	        END_IF;
	    END_REGION

	    REGION UNLOADERS & COOLING CONVEYORS
	        IF (#internal.boManSelOnPressL OR #internal.boSetupSelOnPressL OR #internal.boSetupProcActiveL) AND #internal.panel[#PB_Configuration.itLeftSelPbID].boSelect THEN
	            // Enable push-buttons
	            #internal.panel[#PB_Configuration.itUnloaderPbID].boEnable := TRUE;
	            #internal.panel[#PB_Configuration.itUnloaderPCIPbID].boEnable := TRUE;

	            // Modules fault & warning
	            #internal.panel[#PB_Configuration.itUnloaderPbID].boAborted := #EQunloaderL."to".boStatusAbortedEQ OR #EQunloaderL."to".boStatusAbortedSwingInPress OR #EQunloaderL."to".boStatusAbortedUDMove OR #EQunloaderL."to".boStatusAbortedPaddles;
	            #internal.panel[#PB_Configuration.itUnloaderPbID].boHeld := #EQunloaderL."to".boStatusHeldEQ OR #EQunloaderL."to".boStatusHeldSwingInPress OR #EQunloaderL."to".boStatusHeldUDMove OR #EQunloaderL."to".boStatusHeldPaddles;
	            #internal.panel[#PB_Configuration.itUnloaderPCIPbID].boAborted := #EQunloaderL."to".boStatusAbortedEQ OR #EQunloaderL."to".boStatusAbortedSwingInPci OR #EQunloaderL."to".boStatusAbortedExtend;
	            #internal.panel[#PB_Configuration.itUnloaderPCIPbID].boHeld := #EQunloaderL."to".boStatusHeldEQ OR #EQunloaderL."to".boStatusHeldSwingInPci OR #EQunloaderL."to".boStatusHeldExtend;

	            // Unloaders: manual commands
	            IF #internal.panel[#PB_Configuration.itUnloaderPbID].boSelect THEN
	                #internal.panel[#PB_Configuration.itLeftSelPbID].boAborted := #EQunloaderL."to".boStatusAbortedEQ OR #EQunloaderL."to".boStatusAbortedSwingInPress OR #EQunloaderL."to".boStatusAbortedUDMove OR #EQunloaderL."to".boStatusAbortedPaddles;
	                #internal.panel[#PB_Configuration.itLeftSelPbID].boHeld := #EQunloaderL."to".boStatusHeldEQ OR #EQunloaderL."to".boStatusHeldSwingInPress OR #EQunloaderL."to".boStatusHeldUDMove OR #EQunloaderL."to".boStatusHeldPaddles;

	                #internal.panel[#PB_Configuration.itInCmdPbID].boOnPos := #EQunloaderL."to".boPosSwingIn;
	                #internal.panel[#PB_Configuration.itOutCmdPbID].boOnPos := #EQunloaderL."to".boPosSwingOut;
	                #internal.panel[#PB_Configuration.itUpCmdPbID].boOnPos := #EQunloaderL."to".boPosUnloaderUp;
	                #internal.panel[#PB_Configuration.itDownCmdPbID].boOnPos := #EQunloaderL."to".boPosUnloaderDown;
	                #internal.panel[#PB_Configuration.itRetractCmdPbID].boOnPos := #EQunloaderL."to".boPosPaddlesRet;
	                #internal.panel[#PB_Configuration.itExpandCmdPbID].boOnPos := #EQunloaderL."to".boPosPaddlesExp;

	                #internal.panel[#PB_Configuration.itInCmdPbID].boMoving := #EQunloaderL."to".boMoveSwingIn;
	                #internal.panel[#PB_Configuration.itOutCmdPbID].boMoving := #EQunloaderL."to".boMoveSwingOut;
	                #internal.panel[#PB_Configuration.itUpCmdPbID].boMoving := #EQunloaderL."to".boMoveUnloaderUp;
	                #internal.panel[#PB_Configuration.itDownCmdPbID].boMoving := #EQunloaderL."to".boMoveUnloaderDown;
	                #internal.panel[#PB_Configuration.itRetractCmdPbID].boMoving := #EQunloaderL."to".boMovePaddlesRet;
	                #internal.panel[#PB_Configuration.itExpandCmdPbID].boMoving := #EQunloaderL."to".boMovePaddlesExp;

	                #internal.panel[#PB_Configuration.itInCmdPbID].boEnable := #EQunloaderL."to".boEnaSwingIn OR #internal.panel[#PB_Configuration.itInCmdPbID].boOnPos OR #internal.panel[#PB_Configuration.itInCmdPbID].boMoving;
	                #internal.panel[#PB_Configuration.itOutCmdPbID].boEnable := #EQunloaderL."to".boEnaSwingOut OR #internal.panel[#PB_Configuration.itOutCmdPbID].boOnPos OR #internal.panel[#PB_Configuration.itOutCmdPbID].boMoving;
	                #internal.panel[#PB_Configuration.itUpCmdPbID].boEnable := #EQunloaderL."to".boEnaUnloaderUp OR #internal.panel[#PB_Configuration.itUpCmdPbID].boOnPos OR #internal.panel[#PB_Configuration.itUpCmdPbID].boMoving;
	                #internal.panel[#PB_Configuration.itDownCmdPbID].boEnable := #EQunloaderL."to".boEnaUnloaderDown OR #internal.panel[#PB_Configuration.itDownCmdPbID].boOnPos OR #internal.panel[#PB_Configuration.itDownCmdPbID].boMoving;
	                #internal.panel[#PB_Configuration.itRetractCmdPbID].boEnable := #EQunloaderL."to".boEnaPaddlesRet OR #internal.panel[#PB_Configuration.itRetractCmdPbID].boOnPos OR #internal.panel[#PB_Configuration.itRetractCmdPbID].boMoving;
	                #internal.panel[#PB_Configuration.itExpandCmdPbID].boEnable := #EQunloaderL."to".boEnaPaddlesExp OR #internal.panel[#PB_Configuration.itExpandCmdPbID].boOnPos OR #internal.panel[#PB_Configuration.itExpandCmdPbID].boMoving;

	                #EQunloaderL.from.boCmdSwingIn := #internal.panel[#PB_Configuration.itInCmdPbID].boCmdOn;
	                #EQunloaderL.from.boCmdSwingOut := #internal.panel[#PB_Configuration.itOutCmdPbID].boCmdOn;
	                #EQunloaderL.from.boCmdUDMoveDown := #internal.panel[#PB_Configuration.itDownCmdPbID].boCmdOn;
	                #EQunloaderL.from.boCmdUDMoveUp := #internal.panel[#PB_Configuration.itUpCmdPbID].boCmdOn;
	                #EQunloaderL.from.boCmdPaddlesRet := #internal.panel[#PB_Configuration.itRetractCmdPbID].boCmdOn;
	                #EQunloaderL.from.boCmdPaddlesExp := #internal.panel[#PB_Configuration.itExpandCmdPbID].boCmdOn;
	            END_IF;

	            // Unloaders PCI: manual commands
	            IF #internal.panel[#PB_Configuration.itUnloaderPCIPbID].boSelect THEN
	                #internal.panel[#PB_Configuration.itLeftSelPbID].boAborted := #EQunloaderL."to".boStatusAbortedEQ OR #EQunloaderL."to".boStatusAbortedSwingInPress OR #EQunloaderL."to".boStatusAbortedUDMove OR #EQunloaderL."to".boStatusAbortedPaddles;
	                #internal.panel[#PB_Configuration.itLeftSelPbID].boHeld := #EQunloaderL."to".boStatusHeldEQ OR #EQunloaderL."to".boStatusHeldSwingInPress OR #EQunloaderL."to".boStatusHeldUDMove OR #EQunloaderL."to".boStatusHeldPaddles;

	                #internal.panel[#PB_Configuration.itInCmdPbID].boOnPos := #EQunloaderL."to".boPosExtendRet;
	                #internal.panel[#PB_Configuration.itOutCmdPbID].boOnPos := #EQunloaderL."to".boPosExtendExp;
	                #internal.panel[#PB_Configuration.itUpCmdPbID].boOnPos := #EQunloaderL."to".boPosUnloaderUp;
	                #internal.panel[#PB_Configuration.itDownCmdPbID].boOnPos := #EQunloaderL."to".boPosUnloaderDown;
	                #internal.panel[#PB_Configuration.itRetractCmdPbID].boOnPos := #EQunloaderL."to".boPosPaddlesRet;
	                #internal.panel[#PB_Configuration.itExpandCmdPbID].boOnPos := #EQunloaderL."to".boPosPaddlesExp;

	                #internal.panel[#PB_Configuration.itInCmdPbID].boMoving := #EQunloaderL."to".boMoveExtendRet;
	                #internal.panel[#PB_Configuration.itOutCmdPbID].boMoving := #EQunloaderL."to".boMoveExtendExp;
	                #internal.panel[#PB_Configuration.itUpCmdPbID].boMoving := #EQunloaderL."to".boMoveUnloaderUp;
	                #internal.panel[#PB_Configuration.itDownCmdPbID].boMoving := #EQunloaderL."to".boMoveUnloaderDown;
	                #internal.panel[#PB_Configuration.itRetractCmdPbID].boMoving := #EQunloaderL."to".boMovePaddlesRet;
	                #internal.panel[#PB_Configuration.itExpandCmdPbID].boMoving := #EQunloaderL."to".boMovePaddlesExp;

	                #internal.panel[#PB_Configuration.itInCmdPbID].boEnable := #EQunloaderL."to".boEnaExtendRet OR #internal.panel[#PB_Configuration.itInCmdPbID].boOnPos OR #internal.panel[#PB_Configuration.itInCmdPbID].boMoving;
	                #internal.panel[#PB_Configuration.itOutCmdPbID].boEnable := #EQunloaderL."to".boEnaExtendExp OR #internal.panel[#PB_Configuration.itOutCmdPbID].boOnPos OR #internal.panel[#PB_Configuration.itOutCmdPbID].boMoving;
	                #internal.panel[#PB_Configuration.itUpCmdPbID].boEnable := #EQunloaderL."to".boEnaUnloaderUp OR #internal.panel[#PB_Configuration.itUpCmdPbID].boOnPos OR #internal.panel[#PB_Configuration.itUpCmdPbID].boMoving;
	                #internal.panel[#PB_Configuration.itDownCmdPbID].boEnable := #EQunloaderL."to".boEnaUnloaderDown OR #internal.panel[#PB_Configuration.itDownCmdPbID].boOnPos OR #internal.panel[#PB_Configuration.itDownCmdPbID].boMoving;
	                #internal.panel[#PB_Configuration.itRetractCmdPbID].boEnable := #EQunloaderL."to".boEnaPaddlesRet OR #internal.panel[#PB_Configuration.itRetractCmdPbID].boOnPos OR #internal.panel[#PB_Configuration.itRetractCmdPbID].boMoving;
	                #internal.panel[#PB_Configuration.itExpandCmdPbID].boEnable := #EQunloaderL."to".boEnaPaddlesExp OR #internal.panel[#PB_Configuration.itExpandCmdPbID].boOnPos OR #internal.panel[#PB_Configuration.itExpandCmdPbID].boMoving;

	                #EQunloaderL.from.boCmdExtendRet := #internal.panel[#PB_Configuration.itInCmdPbID].boCmdOn;
	                #EQunloaderL.from.boCmdExtendExp := #internal.panel[#PB_Configuration.itOutCmdPbID].boCmdOn;
	                #EQunloaderL.from.boCmdUDMoveDown := #internal.panel[#PB_Configuration.itDownCmdPbID].boCmdOn;
	                #EQunloaderL.from.boCmdUDMoveUp := #internal.panel[#PB_Configuration.itUpCmdPbID].boCmdOn;
	                #EQunloaderL.from.boCmdPaddlesRet := #internal.panel[#PB_Configuration.itRetractCmdPbID].boCmdOn;
	                #EQunloaderL.from.boCmdPaddlesExp := #internal.panel[#PB_Configuration.itExpandCmdPbID].boCmdOn;
	            END_IF;
	        END_IF;
	        IF (#internal.boManSelOnExitConvL OR #internal.boSetupSelOnExitConvL OR #internal.boSetupProcActiveL) AND #internal.panel[#PB_Configuration.itLeftSelPbID].boSelect THEN
	            // Enable push-buttons
	            #internal.panel[#PB_Configuration.itExitConvPbId].boEnable := TRUE;

	            // Modules fault & warning
	            #internal.panel[#PB_Configuration.itExitConvPbId].boAborted := #EQExitConvL."to".boStatusAbortedEQ OR #EQExitConvL."to".boStatusAbortedLwConveyor OR #EQExitConvL."to".boStatusAbortedLwBlocks;
	            #internal.panel[#PB_Configuration.itExitConvPbId].boHeld := #EQExitConvL."to".boStatusHeldEQ OR #EQExitConvL."to".boStatusHeldLwConveyor OR #EQExitConvL."to".boStatusHeldLwBlocks;

	            // Cooling Conveyors : manual commands
	            IF #internal.panel[#PB_Configuration.itExitConvPbId].boSelect THEN
	                #internal.panel[#PB_Configuration.itLeftSelPbID].boAborted := #EQExitConvL."to".boStatusAbortedEQ OR #EQExitConvL."to".boStatusAbortedLwConveyor OR #EQExitConvL."to".boStatusAbortedLwBlocks;
	                #internal.panel[#PB_Configuration.itLeftSelPbID].boHeld := #EQExitConvL."to".boStatusHeldEQ OR #EQExitConvL."to".boStatusHeldLwConveyor OR #EQExitConvL."to".boStatusHeldLwBlocks;

	                #internal.panel[#PB_Configuration.itUpCmdPbID].boOnPos := #EQExitConvL."to".boPosConveyorUp;
	                #internal.panel[#PB_Configuration.itDownCmdPbID].boOnPos := #EQExitConvL."to".boPosConveyorDown;
	                #internal.panel[#PB_Configuration.itOutCmdPbID].boOnPos := FALSE;
	                #internal.panel[#PB_Configuration.itLockCmdPbID].boOnPos := #EQExitConvL."to".boPosBlockIns;
	                #internal.panel[#PB_Configuration.itUnlockCmdPbID].boOnPos := #EQExitConvL."to".boPosBlockRel;

	                #internal.panel[#PB_Configuration.itUpCmdPbID].boMoving := #EQExitConvL."to".boMoveConveyorUp;
	                #internal.panel[#PB_Configuration.itDownCmdPbID].boMoving := #EQExitConvL."to".boMoveConveyorDown;
	                #internal.panel[#PB_Configuration.itOutCmdPbID].boMoving := #EQExitConvL."to".boMoveConveyorFwd;
	                #internal.panel[#PB_Configuration.itLockCmdPbID].boMoving := #EQExitConvL."to".boMoveBlockIns;
	                #internal.panel[#PB_Configuration.itUnlockCmdPbID].boMoving := #EQExitConvL."to".boMoveBlockRel;

	                #internal.panel[#PB_Configuration.itUpCmdPbID].boEnable := #EQExitConvL."to".boEnaConveyorUp OR #internal.panel[#PB_Configuration.itInCmdPbID].boOnPos OR #internal.panel[#PB_Configuration.itInCmdPbID].boMoving;
	                #internal.panel[#PB_Configuration.itDownCmdPbID].boEnable := #EQExitConvL."to".boEnaConveyorDown OR #internal.panel[#PB_Configuration.itInCmdPbID].boOnPos OR #internal.panel[#PB_Configuration.itInCmdPbID].boMoving;
	                #internal.panel[#PB_Configuration.itOutCmdPbID].boEnable := #EQExitConvL."to".boEnaConveyorFwd OR #internal.panel[#PB_Configuration.itInCmdPbID].boOnPos OR #internal.panel[#PB_Configuration.itInCmdPbID].boMoving;
	                #internal.panel[#PB_Configuration.itLockCmdPbID].boEnable := #EQExitConvL."to".boEnaBlockIns OR #internal.panel[#PB_Configuration.itInCmdPbID].boOnPos OR #internal.panel[#PB_Configuration.itInCmdPbID].boMoving;
	                #internal.panel[#PB_Configuration.itUnlockCmdPbID].boEnable := #EQExitConvL."to".boEnaBlockRel OR #internal.panel[#PB_Configuration.itInCmdPbID].boOnPos OR #internal.panel[#PB_Configuration.itInCmdPbID].boMoving;

	                #EQExitConvL.from.boCmdConveyorUp := #internal.panel[#PB_Configuration.itUpCmdPbID].boCmdOn;
	                #EQExitConvL.from.boCmdConveyorDown := #internal.panel[#PB_Configuration.itDownCmdPbID].boCmdOn;
	                #EQExitConvL.from.boCmdConveyorFwd := #internal.panel[#PB_Configuration.itOutCmdPbID].boCmdOn;
	                #EQExitConvL.from.boCmdBlockIns := #internal.panel[#PB_Configuration.itLockCmdPbID].boCmdOn;
	                #EQExitConvL.from.boCmdBlockRel := #internal.panel[#PB_Configuration.itUnlockCmdPbID].boCmdOn;
	            END_IF;
	        END_IF;

	        IF (#internal.boManSelOnPressR OR #internal.boSetupSelOnPressR OR #internal.boSetupProcActiveR) AND #internal.panel[#PB_Configuration.itRightSelPbID].boSelect THEN
	            // Enable push-buttons
	            #internal.panel[#PB_Configuration.itUnloaderPbID].boEnable := TRUE;
	            #internal.panel[#PB_Configuration.itUnloaderPCIPbID].boEnable := TRUE;

	            // Modules fault & warning
	            #internal.panel[#PB_Configuration.itUnloaderPbID].boAborted := #EQunloaderR."to".boStatusAbortedEQ OR #EQunloaderR."to".boStatusAbortedSwingInPress OR #EQunloaderR."to".boStatusAbortedUDMove OR #EQunloaderR."to".boStatusAbortedPaddles;
	            #internal.panel[#PB_Configuration.itUnloaderPbID].boHeld := #EQunloaderR."to".boStatusHeldEQ OR #EQunloaderR."to".boStatusHeldSwingInPress OR #EQunloaderR."to".boStatusHeldUDMove OR #EQunloaderR."to".boStatusHeldPaddles;
	            #internal.panel[#PB_Configuration.itUnloaderPCIPbID].boAborted := #EQunloaderR."to".boStatusAbortedEQ OR #EQunloaderR."to".boStatusAbortedSwingInPci OR #EQunloaderR."to".boStatusAbortedExtend;
	            #internal.panel[#PB_Configuration.itUnloaderPCIPbID].boHeld := #EQunloaderR."to".boStatusHeldEQ OR #EQunloaderR."to".boStatusHeldSwingInPci OR #EQunloaderR."to".boStatusHeldExtend;

	            // Unloaders: manual commands
	            IF #internal.panel[#PB_Configuration.itUnloaderPbID].boSelect THEN
	                #internal.panel[#PB_Configuration.itRightSelPbID].boAborted := #EQunloaderR."to".boStatusAbortedEQ OR #EQunloaderR."to".boStatusAbortedSwingInPress OR #EQunloaderR."to".boStatusAbortedUDMove OR #EQunloaderR."to".boStatusAbortedPaddles;
	                #internal.panel[#PB_Configuration.itRightSelPbID].boHeld := #EQunloaderR."to".boStatusHeldEQ OR #EQunloaderR."to".boStatusHeldSwingInPress OR #EQunloaderR."to".boStatusHeldUDMove OR #EQunloaderR."to".boStatusHeldPaddles;

	                #internal.panel[#PB_Configuration.itInCmdPbID].boOnPos := #EQunloaderR."to".boPosSwingIn;
	                #internal.panel[#PB_Configuration.itOutCmdPbID].boOnPos := #EQunloaderR."to".boPosSwingOut;
	                #internal.panel[#PB_Configuration.itUpCmdPbID].boOnPos := #EQunloaderR."to".boPosUnloaderUp;
	                #internal.panel[#PB_Configuration.itDownCmdPbID].boOnPos := #EQunloaderR."to".boPosUnloaderDown;
	                #internal.panel[#PB_Configuration.itRetractCmdPbID].boOnPos := #EQunloaderR."to".boPosPaddlesRet;
	                #internal.panel[#PB_Configuration.itExpandCmdPbID].boOnPos := #EQunloaderR."to".boPosPaddlesExp;

	                #internal.panel[#PB_Configuration.itInCmdPbID].boMoving := #EQunloaderR."to".boMoveSwingIn;
	                #internal.panel[#PB_Configuration.itOutCmdPbID].boMoving := #EQunloaderR."to".boMoveSwingOut;
	                #internal.panel[#PB_Configuration.itUpCmdPbID].boMoving := #EQunloaderR."to".boMoveUnloaderUp;
	                #internal.panel[#PB_Configuration.itDownCmdPbID].boMoving := #EQunloaderR."to".boMoveUnloaderDown;
	                #internal.panel[#PB_Configuration.itRetractCmdPbID].boMoving := #EQunloaderR."to".boMovePaddlesRet;
	                #internal.panel[#PB_Configuration.itExpandCmdPbID].boMoving := #EQunloaderR."to".boMovePaddlesExp;

	                #internal.panel[#PB_Configuration.itInCmdPbID].boEnable := #EQunloaderR."to".boEnaSwingIn OR #internal.panel[#PB_Configuration.itInCmdPbID].boOnPos OR #internal.panel[#PB_Configuration.itInCmdPbID].boMoving;
	                #internal.panel[#PB_Configuration.itOutCmdPbID].boEnable := #EQunloaderR."to".boEnaSwingOut OR #internal.panel[#PB_Configuration.itOutCmdPbID].boOnPos OR #internal.panel[#PB_Configuration.itOutCmdPbID].boMoving;
	                #internal.panel[#PB_Configuration.itUpCmdPbID].boEnable := #EQunloaderR."to".boEnaUnloaderUp OR #internal.panel[#PB_Configuration.itUpCmdPbID].boOnPos OR #internal.panel[#PB_Configuration.itUpCmdPbID].boMoving;
	                #internal.panel[#PB_Configuration.itDownCmdPbID].boEnable := #EQunloaderR."to".boEnaUnloaderDown OR #internal.panel[#PB_Configuration.itDownCmdPbID].boOnPos OR #internal.panel[#PB_Configuration.itDownCmdPbID].boMoving;
	                #internal.panel[#PB_Configuration.itRetractCmdPbID].boEnable := #EQunloaderR."to".boEnaPaddlesRet OR #internal.panel[#PB_Configuration.itRetractCmdPbID].boOnPos OR #internal.panel[#PB_Configuration.itRetractCmdPbID].boMoving;
	                #internal.panel[#PB_Configuration.itExpandCmdPbID].boEnable := #EQunloaderR."to".boEnaPaddlesExp OR #internal.panel[#PB_Configuration.itExpandCmdPbID].boOnPos OR #internal.panel[#PB_Configuration.itExpandCmdPbID].boMoving;

	                #EQunloaderR.from.boCmdSwingIn := #internal.panel[#PB_Configuration.itInCmdPbID].boCmdOn;
	                #EQunloaderR.from.boCmdSwingOut := #internal.panel[#PB_Configuration.itOutCmdPbID].boCmdOn;
	                #EQunloaderR.from.boCmdUDMoveDown := #internal.panel[#PB_Configuration.itDownCmdPbID].boCmdOn;
	                #EQunloaderR.from.boCmdUDMoveUp := #internal.panel[#PB_Configuration.itUpCmdPbID].boCmdOn;
	                #EQunloaderR.from.boCmdPaddlesRet := #internal.panel[#PB_Configuration.itRetractCmdPbID].boCmdOn;
	                #EQunloaderR.from.boCmdPaddlesExp := #internal.panel[#PB_Configuration.itExpandCmdPbID].boCmdOn;
	            END_IF;

	            // Unloaders PCI: manual commands
	            IF #internal.panel[#PB_Configuration.itUnloaderPCIPbID].boSelect THEN
	                #internal.panel[#PB_Configuration.itRightSelPbID].boAborted := #EQunloaderR."to".boStatusAbortedEQ OR #EQunloaderR."to".boStatusAbortedSwingInPci OR #EQunloaderR."to".boStatusAbortedExtend;
	                #internal.panel[#PB_Configuration.itRightSelPbID].boHeld := #EQunloaderR."to".boStatusHeldEQ OR #EQunloaderR."to".boStatusHeldSwingInPci OR #EQunloaderR."to".boStatusHeldExtend;

	                #internal.panel[#PB_Configuration.itInCmdPbID].boOnPos := #EQunloaderR."to".boPosExtendRet;
	                #internal.panel[#PB_Configuration.itOutCmdPbID].boOnPos := #EQunloaderR."to".boPosExtendExp;
	                #internal.panel[#PB_Configuration.itUpCmdPbID].boOnPos := #EQunloaderR."to".boPosUnloaderUp;
	                #internal.panel[#PB_Configuration.itDownCmdPbID].boOnPos := #EQunloaderR."to".boPosUnloaderDown;
	                #internal.panel[#PB_Configuration.itRetractCmdPbID].boOnPos := #EQunloaderR."to".boPosPaddlesRet;
	                #internal.panel[#PB_Configuration.itExpandCmdPbID].boOnPos := #EQunloaderR."to".boPosPaddlesExp;

	                #internal.panel[#PB_Configuration.itInCmdPbID].boMoving := #EQunloaderR."to".boMoveExtendRet;
	                #internal.panel[#PB_Configuration.itOutCmdPbID].boMoving := #EQunloaderR."to".boMoveExtendExp;
	                #internal.panel[#PB_Configuration.itUpCmdPbID].boMoving := #EQunloaderR."to".boMoveUnloaderUp;
	                #internal.panel[#PB_Configuration.itDownCmdPbID].boMoving := #EQunloaderR."to".boMoveUnloaderDown;
	                #internal.panel[#PB_Configuration.itRetractCmdPbID].boMoving := #EQunloaderR."to".boMovePaddlesRet;
	                #internal.panel[#PB_Configuration.itExpandCmdPbID].boMoving := #EQunloaderR."to".boMovePaddlesExp;

	                #internal.panel[#PB_Configuration.itInCmdPbID].boEnable := #EQunloaderR."to".boEnaExtendRet OR #internal.panel[#PB_Configuration.itInCmdPbID].boOnPos OR #internal.panel[#PB_Configuration.itInCmdPbID].boMoving;
	                #internal.panel[#PB_Configuration.itOutCmdPbID].boEnable := #EQunloaderR."to".boEnaExtendExp OR #internal.panel[#PB_Configuration.itOutCmdPbID].boOnPos OR #internal.panel[#PB_Configuration.itOutCmdPbID].boMoving;
	                #internal.panel[#PB_Configuration.itUpCmdPbID].boEnable := #EQunloaderR."to".boEnaUnloaderUp OR #internal.panel[#PB_Configuration.itUpCmdPbID].boOnPos OR #internal.panel[#PB_Configuration.itUpCmdPbID].boMoving;
	                #internal.panel[#PB_Configuration.itDownCmdPbID].boEnable := #EQunloaderR."to".boEnaUnloaderDown OR #internal.panel[#PB_Configuration.itDownCmdPbID].boOnPos OR #internal.panel[#PB_Configuration.itDownCmdPbID].boMoving;
	                #internal.panel[#PB_Configuration.itRetractCmdPbID].boEnable := #EQunloaderR."to".boEnaPaddlesRet OR #internal.panel[#PB_Configuration.itRetractCmdPbID].boOnPos OR #internal.panel[#PB_Configuration.itRetractCmdPbID].boMoving;
	                #internal.panel[#PB_Configuration.itExpandCmdPbID].boEnable := #EQunloaderR."to".boEnaPaddlesExp OR #internal.panel[#PB_Configuration.itExpandCmdPbID].boOnPos OR #internal.panel[#PB_Configuration.itExpandCmdPbID].boMoving;

	                #EQunloaderR.from.boCmdExtendRet := #internal.panel[#PB_Configuration.itInCmdPbID].boCmdOn;
	                #EQunloaderR.from.boCmdExtendExp := #internal.panel[#PB_Configuration.itOutCmdPbID].boCmdOn;
	                #EQunloaderR.from.boCmdUDMoveDown := #internal.panel[#PB_Configuration.itDownCmdPbID].boCmdOn;
	                #EQunloaderR.from.boCmdUDMoveUp := #internal.panel[#PB_Configuration.itUpCmdPbID].boCmdOn;
	                #EQunloaderR.from.boCmdPaddlesRet := #internal.panel[#PB_Configuration.itRetractCmdPbID].boCmdOn;
	                #EQunloaderR.from.boCmdPaddlesExp := #internal.panel[#PB_Configuration.itExpandCmdPbID].boCmdOn;
	            END_IF;
	        END_IF;
	        IF (#internal.boManSelOnExitConvR OR #internal.boSetupSelOnExitConvR OR #internal.boSetupProcActiveR) AND #internal.panel[#PB_Configuration.itRightSelPbID].boSelect THEN

	            // Enable push-buttons
	            #internal.panel[#PB_Configuration.itExitConvPbId].boEnable := TRUE;

	            // Modules fault & warning
	            #internal.panel[#PB_Configuration.itExitConvPbId].boAborted := #EQExitConvR."to".boStatusAbortedEQ OR #EQExitConvR."to".boStatusAbortedLwConveyor OR #EQExitConvR."to".boStatusAbortedLwBlocks;
	            #internal.panel[#PB_Configuration.itExitConvPbId].boHeld := #EQExitConvR."to".boStatusHeldEQ OR #EQExitConvR."to".boStatusHeldLwConveyor OR #EQExitConvR."to".boStatusHeldLwBlocks;

	            // Cooling Conveyors : manual commands
	            IF #internal.panel[#PB_Configuration.itExitConvPbId].boSelect THEN
	                #internal.panel[#PB_Configuration.itRightSelPbID].boAborted := #EQExitConvR."to".boStatusAbortedEQ OR #EQExitConvR."to".boStatusAbortedLwConveyor OR #EQExitConvR."to".boStatusAbortedLwBlocks;
	                #internal.panel[#PB_Configuration.itRightSelPbID].boHeld := #EQExitConvR."to".boStatusHeldEQ OR #EQExitConvR."to".boStatusHeldLwConveyor OR #EQExitConvR."to".boStatusHeldLwBlocks;

	                #internal.panel[#PB_Configuration.itUpCmdPbID].boOnPos := #EQExitConvR."to".boPosConveyorUp;
	                #internal.panel[#PB_Configuration.itDownCmdPbID].boOnPos := #EQExitConvR."to".boPosConveyorDown;
	                #internal.panel[#PB_Configuration.itOutCmdPbID].boOnPos := FALSE;
	                #internal.panel[#PB_Configuration.itLockCmdPbID].boOnPos := #EQExitConvR."to".boPosBlockIns;
	                #internal.panel[#PB_Configuration.itUnlockCmdPbID].boOnPos := #EQExitConvR."to".boPosBlockRel;

	                #internal.panel[#PB_Configuration.itUpCmdPbID].boMoving := #EQExitConvR."to".boMoveConveyorUp;
	                #internal.panel[#PB_Configuration.itDownCmdPbID].boMoving := #EQExitConvR."to".boMoveConveyorDown;
	                #internal.panel[#PB_Configuration.itOutCmdPbID].boMoving := #EQExitConvR."to".boMoveConveyorFwd;
	                #internal.panel[#PB_Configuration.itLockCmdPbID].boMoving := #EQExitConvR."to".boMoveBlockIns;
	                #internal.panel[#PB_Configuration.itUnlockCmdPbID].boMoving := #EQExitConvR."to".boMoveBlockRel;

	                #internal.panel[#PB_Configuration.itUpCmdPbID].boEnable := #EQExitConvR."to".boEnaConveyorUp OR #internal.panel[#PB_Configuration.itInCmdPbID].boOnPos OR #internal.panel[#PB_Configuration.itInCmdPbID].boMoving;
	                #internal.panel[#PB_Configuration.itDownCmdPbID].boEnable := #EQExitConvR."to".boEnaConveyorDown OR #internal.panel[#PB_Configuration.itInCmdPbID].boOnPos OR #internal.panel[#PB_Configuration.itInCmdPbID].boMoving;
	                #internal.panel[#PB_Configuration.itOutCmdPbID].boEnable := #EQExitConvR."to".boEnaConveyorFwd OR #internal.panel[#PB_Configuration.itInCmdPbID].boOnPos OR #internal.panel[#PB_Configuration.itInCmdPbID].boMoving;
	                #internal.panel[#PB_Configuration.itLockCmdPbID].boEnable := #EQExitConvR."to".boEnaBlockIns OR #internal.panel[#PB_Configuration.itInCmdPbID].boOnPos OR #internal.panel[#PB_Configuration.itInCmdPbID].boMoving;
	                #internal.panel[#PB_Configuration.itUnlockCmdPbID].boEnable := #EQExitConvR."to".boEnaBlockRel OR #internal.panel[#PB_Configuration.itInCmdPbID].boOnPos OR #internal.panel[#PB_Configuration.itInCmdPbID].boMoving;

	                #EQExitConvR.from.boCmdConveyorUp := #internal.panel[#PB_Configuration.itUpCmdPbID].boCmdOn;
	                #EQExitConvR.from.boCmdConveyorDown := #internal.panel[#PB_Configuration.itDownCmdPbID].boCmdOn;
	                #EQExitConvR.from.boCmdConveyorFwd := #internal.panel[#PB_Configuration.itOutCmdPbID].boCmdOn;
	                #EQExitConvR.from.boCmdBlockIns := #internal.panel[#PB_Configuration.itLockCmdPbID].boCmdOn;
	                #EQExitConvR.from.boCmdBlockRel := #internal.panel[#PB_Configuration.itUnlockCmdPbID].boCmdOn;
	            END_IF;

	        END_IF;

	        IF ((#internal.boManSelOnPressL OR #internal.boSetupSelOnPressL OR #internal.boSetupProcActiveL) AND #internal.panel[#PB_Configuration.itLeftSelPbID].boSelect) AND
	            ((#internal.boManSelOnPressR OR #internal.boSetupSelOnPressR OR #internal.boSetupProcActiveR) AND #internal.panel[#PB_Configuration.itRightSelPbID].boSelect) THEN
	            // Enable push-buttons
	            #internal.panel[#PB_Configuration.itUnloaderPbID].boEnable := TRUE;
	            #internal.panel[#PB_Configuration.itUnloaderPCIPbID].boEnable := TRUE;

	            // Modules fault & warning
	            #internal.panel[#PB_Configuration.itUnloaderPbID].boAborted := #EQunloaderL."to".boStatusAbortedEQ OR #EQunloaderL."to".boStatusAbortedSwingInPress OR #EQunloaderL."to".boStatusAbortedUDMove OR #EQunloaderL."to".boStatusAbortedPaddles OR
	            #EQunloaderR."to".boStatusAbortedEQ OR #EQunloaderR."to".boStatusAbortedSwingInPress OR #EQunloaderR."to".boStatusAbortedUDMove OR #EQunloaderR."to".boStatusAbortedPaddles;
	            #internal.panel[#PB_Configuration.itUnloaderPbID].boHeld := #EQunloaderL."to".boStatusHeldEQ OR #EQunloaderL."to".boStatusHeldSwingInPress OR #EQunloaderL."to".boStatusHeldUDMove OR #EQunloaderL."to".boStatusHeldPaddles OR
	            #EQunloaderR."to".boStatusHeldEQ OR #EQunloaderR."to".boStatusHeldSwingInPress OR #EQunloaderR."to".boStatusHeldUDMove OR #EQunloaderR."to".boStatusHeldPaddles;

	            #internal.panel[#PB_Configuration.itUnloaderPCIPbID].boAborted := #EQunloaderL."to".boStatusAbortedEQ OR #EQunloaderL."to".boStatusAbortedSwingInPci OR #EQunloaderL."to".boStatusAbortedExtend OR
	            #EQunloaderR."to".boStatusAbortedEQ OR #EQunloaderR."to".boStatusAbortedSwingInPci OR #EQunloaderR."to".boStatusAbortedExtend;
	            #internal.panel[#PB_Configuration.itUnloaderPCIPbID].boHeld := #EQunloaderL."to".boStatusHeldEQ OR #EQunloaderL."to".boStatusHeldSwingInPci OR #EQunloaderL."to".boStatusHeldExtend OR
	            #EQunloaderR."to".boStatusHeldEQ OR #EQunloaderR."to".boStatusHeldSwingInPci OR #EQunloaderR."to".boStatusHeldExtend;

	            // Unloaders: manual commands
	            IF #internal.panel[#PB_Configuration.itUnloaderPbID].boSelect THEN
	                #internal.panel[#PB_Configuration.itInCmdPbID].boOnPos := #EQunloaderL."to".boPosSwingIn AND #EQunloaderR."to".boPosSwingIn;
	                #internal.panel[#PB_Configuration.itOutCmdPbID].boOnPos := #EQunloaderL."to".boPosSwingOut AND #EQunloaderR."to".boPosSwingOut;
	                #internal.panel[#PB_Configuration.itUpCmdPbID].boOnPos := #EQunloaderL."to".boPosUnloaderUp AND #EQunloaderR."to".boPosUnloaderUp;
	                #internal.panel[#PB_Configuration.itDownCmdPbID].boOnPos := #EQunloaderL."to".boPosUnloaderDown AND #EQunloaderR."to".boPosUnloaderDown;
	                #internal.panel[#PB_Configuration.itRetractCmdPbID].boOnPos := #EQunloaderL."to".boPosPaddlesRet AND #EQunloaderR."to".boPosPaddlesRet;
	                #internal.panel[#PB_Configuration.itExpandCmdPbID].boOnPos := #EQunloaderL."to".boPosPaddlesExp AND #EQunloaderR."to".boPosPaddlesExp;

	                #internal.panel[#PB_Configuration.itInCmdPbID].boMoving := #EQunloaderL."to".boMoveSwingIn AND #EQunloaderR."to".boMoveSwingIn;
	                #internal.panel[#PB_Configuration.itOutCmdPbID].boMoving := #EQunloaderL."to".boMoveSwingOut AND #EQunloaderR."to".boMoveSwingOut;
	                #internal.panel[#PB_Configuration.itUpCmdPbID].boMoving := #EQunloaderL."to".boMoveUnloaderUp AND #EQunloaderR."to".boMoveUnloaderUp;
	                #internal.panel[#PB_Configuration.itDownCmdPbID].boMoving := #EQunloaderL."to".boMoveUnloaderDown AND #EQunloaderR."to".boMoveUnloaderDown;
	                #internal.panel[#PB_Configuration.itRetractCmdPbID].boMoving := #EQunloaderL."to".boMovePaddlesRet AND #EQunloaderR."to".boMovePaddlesRet;
	                #internal.panel[#PB_Configuration.itExpandCmdPbID].boMoving := #EQunloaderL."to".boMovePaddlesExp AND #EQunloaderR."to".boMovePaddlesExp;

	                #internal.panel[#PB_Configuration.itInCmdPbID].boEnable := #EQunloaderL."to".boEnaSwingIn OR #EQunloaderR."to".boEnaSwingIn OR #internal.panel[#PB_Configuration.itInCmdPbID].boOnPos OR #internal.panel[#PB_Configuration.itInCmdPbID].boMoving;
	                #internal.panel[#PB_Configuration.itOutCmdPbID].boEnable := #EQunloaderL."to".boEnaSwingOut OR #EQunloaderR."to".boEnaSwingOut OR #internal.panel[#PB_Configuration.itOutCmdPbID].boOnPos OR #internal.panel[#PB_Configuration.itOutCmdPbID].boMoving;
	                #internal.panel[#PB_Configuration.itUpCmdPbID].boEnable := #EQunloaderL."to".boEnaUnloaderUp OR #EQunloaderR."to".boEnaUnloaderUp OR #internal.panel[#PB_Configuration.itUpCmdPbID].boOnPos OR #internal.panel[#PB_Configuration.itUpCmdPbID].boMoving;
	                #internal.panel[#PB_Configuration.itDownCmdPbID].boEnable := #EQunloaderL."to".boEnaUnloaderDown OR #EQunloaderR."to".boEnaUnloaderDown OR #internal.panel[#PB_Configuration.itDownCmdPbID].boOnPos OR #internal.panel[#PB_Configuration.itDownCmdPbID].boMoving;
	                #internal.panel[#PB_Configuration.itRetractCmdPbID].boEnable := #EQunloaderL."to".boEnaPaddlesRet OR #EQunloaderR."to".boEnaPaddlesRet OR #internal.panel[#PB_Configuration.itRetractCmdPbID].boOnPos OR #internal.panel[#PB_Configuration.itRetractCmdPbID].boMoving;
	                #internal.panel[#PB_Configuration.itExpandCmdPbID].boEnable := #EQunloaderL."to".boEnaPaddlesExp OR #EQunloaderR."to".boEnaPaddlesExp OR #internal.panel[#PB_Configuration.itExpandCmdPbID].boOnPos OR #internal.panel[#PB_Configuration.itExpandCmdPbID].boMoving;
	            END_IF;

	            // Unloaders PCI: manual commands
	            IF #internal.panel[#PB_Configuration.itUnloaderPCIPbID].boSelect THEN
	                #internal.panel[#PB_Configuration.itInCmdPbID].boOnPos := #EQunloaderL."to".boPosExtendRet AND #EQunloaderR."to".boPosExtendRet;
	                #internal.panel[#PB_Configuration.itOutCmdPbID].boOnPos := #EQunloaderL."to".boPosExtendExp AND #EQunloaderR."to".boPosExtendExp;
	                #internal.panel[#PB_Configuration.itUpCmdPbID].boOnPos := #EQunloaderL."to".boPosUnloaderUp AND #EQunloaderR."to".boPosUnloaderUp;
	                #internal.panel[#PB_Configuration.itDownCmdPbID].boOnPos := #EQunloaderL."to".boPosUnloaderDown AND #EQunloaderR."to".boPosUnloaderDown;
	                #internal.panel[#PB_Configuration.itRetractCmdPbID].boOnPos := #EQunloaderL."to".boPosPaddlesRet AND #EQunloaderR."to".boPosPaddlesRet;
	                #internal.panel[#PB_Configuration.itExpandCmdPbID].boOnPos := #EQunloaderL."to".boPosPaddlesExp AND #EQunloaderR."to".boPosPaddlesExp;

	                #internal.panel[#PB_Configuration.itInCmdPbID].boMoving := #EQunloaderL."to".boMoveExtendRet OR #EQunloaderR."to".boMoveExtendRet;
	                #internal.panel[#PB_Configuration.itOutCmdPbID].boMoving := #EQunloaderL."to".boMoveExtendExp OR #EQunloaderR."to".boMoveExtendExp;
	                #internal.panel[#PB_Configuration.itUpCmdPbID].boMoving := #EQunloaderL."to".boMoveUnloaderUp AND #EQunloaderR."to".boMoveUnloaderUp;
	                #internal.panel[#PB_Configuration.itDownCmdPbID].boMoving := #EQunloaderL."to".boMoveUnloaderDown AND #EQunloaderR."to".boMoveUnloaderDown;
	                #internal.panel[#PB_Configuration.itRetractCmdPbID].boMoving := #EQunloaderL."to".boMovePaddlesRet OR #EQunloaderR."to".boMovePaddlesRet;
	                #internal.panel[#PB_Configuration.itExpandCmdPbID].boMoving := #EQunloaderL."to".boMovePaddlesExp OR #EQunloaderR."to".boMovePaddlesExp;

	                #internal.panel[#PB_Configuration.itInCmdPbID].boEnable := #EQunloaderL."to".boEnaExtendRet OR #EQunloaderR."to".boEnaExtendRet OR #internal.panel[#PB_Configuration.itInCmdPbID].boOnPos OR #internal.panel[#PB_Configuration.itInCmdPbID].boMoving;
	                #internal.panel[#PB_Configuration.itOutCmdPbID].boEnable := #EQunloaderL."to".boEnaExtendExp OR #EQunloaderR."to".boEnaExtendExp OR #internal.panel[#PB_Configuration.itOutCmdPbID].boOnPos OR #internal.panel[#PB_Configuration.itOutCmdPbID].boMoving;
	                #internal.panel[#PB_Configuration.itUpCmdPbID].boEnable := #EQunloaderL."to".boEnaUnloaderUp OR #EQunloaderR."to".boEnaUnloaderUp OR #internal.panel[#PB_Configuration.itUpCmdPbID].boOnPos OR #internal.panel[#PB_Configuration.itUpCmdPbID].boMoving;
	                #internal.panel[#PB_Configuration.itDownCmdPbID].boEnable := #EQunloaderL."to".boEnaUnloaderDown OR #EQunloaderR."to".boEnaUnloaderDown OR #internal.panel[#PB_Configuration.itDownCmdPbID].boOnPos OR #internal.panel[#PB_Configuration.itDownCmdPbID].boMoving;
	                #internal.panel[#PB_Configuration.itRetractCmdPbID].boEnable := #EQunloaderL."to".boEnaPaddlesRet OR #EQunloaderR."to".boEnaPaddlesRet OR #internal.panel[#PB_Configuration.itRetractCmdPbID].boOnPos OR #internal.panel[#PB_Configuration.itRetractCmdPbID].boMoving;
	                #internal.panel[#PB_Configuration.itExpandCmdPbID].boEnable := #EQunloaderL."to".boEnaPaddlesExp OR #EQunloaderR."to".boEnaPaddlesExp OR #internal.panel[#PB_Configuration.itExpandCmdPbID].boOnPos OR #internal.panel[#PB_Configuration.itExpandCmdPbID].boMoving;
	            END_IF;


	            // Enable push-buttons
	            #internal.panel[#PB_Configuration.itExitConvPbId].boEnable := TRUE;

	            // Modules fault & warning
	            #internal.panel[#PB_Configuration.itExitConvPbId].boAborted := #EQExitConvL."to".boStatusAbortedEQ OR #EQExitConvL."to".boStatusAbortedLwConveyor OR #EQExitConvL."to".boStatusAbortedLwBlocks OR
	            #EQExitConvR."to".boStatusAbortedEQ OR #EQExitConvR."to".boStatusAbortedLwConveyor OR #EQExitConvR."to".boStatusAbortedLwBlocks;
	            #internal.panel[#PB_Configuration.itExitConvPbId].boHeld := #EQExitConvL."to".boStatusHeldEQ OR #EQExitConvL."to".boStatusHeldLwConveyor OR #EQExitConvL."to".boStatusHeldLwBlocks OR
	            #EQExitConvR."to".boStatusHeldEQ OR #EQExitConvR."to".boStatusHeldLwConveyor OR #EQExitConvR."to".boStatusHeldLwBlocks;

	            // Cooling Conveyors : manual commands
	            IF #internal.panel[#PB_Configuration.itExitConvPbId].boSelect THEN
	                #internal.panel[#PB_Configuration.itRightSelPbID].boAborted := #EQExitConvL."to".boStatusAbortedEQ OR #EQExitConvL."to".boStatusAbortedLwConveyor OR #EQExitConvL."to".boStatusAbortedLwBlocks OR
	                #EQExitConvR."to".boStatusAbortedEQ OR #EQExitConvR."to".boStatusAbortedLwConveyor OR #EQExitConvR."to".boStatusAbortedLwBlocks;
	                #internal.panel[#PB_Configuration.itRightSelPbID].boHeld := #EQExitConvL."to".boStatusHeldEQ OR #EQExitConvL."to".boStatusHeldLwConveyor OR #EQExitConvL."to".boStatusHeldLwBlocks OR
	                #EQExitConvR."to".boStatusHeldEQ OR #EQExitConvR."to".boStatusHeldLwConveyor OR #EQExitConvR."to".boStatusHeldLwBlocks;

	                #internal.panel[#PB_Configuration.itUpCmdPbID].boOnPos := #EQExitConvL."to".boPosConveyorUp AND #EQExitConvR."to".boPosLwConveyorUp;
	                #internal.panel[#PB_Configuration.itDownCmdPbID].boOnPos := #EQExitConvL."to".boPosConveyorDown AND #EQExitConvR."to".boPosLwConveyorDown;
	                #internal.panel[#PB_Configuration.itOutCmdPbID].boOnPos := FALSE;
	                #internal.panel[#PB_Configuration.itLockCmdPbID].boOnPos := #EQExitConvL."to".boPosBlockIns AND #EQExitConvR."to".boPosLwBlockIns;
	                #internal.panel[#PB_Configuration.itUnlockCmdPbID].boOnPos := #EQExitConvL."to".boPosBlockRel AND #EQExitConvR."to".boPosLwBlockRel;

	                #internal.panel[#PB_Configuration.itUpCmdPbID].boMoving := #EQExitConvR."to".boMoveConveyorUp OR #EQExitConvR."to".boMoveLwConveyorUp;
	                #internal.panel[#PB_Configuration.itDownCmdPbID].boMoving := #EQExitConvR."to".boMoveConveyorDown OR #EQExitConvR."to".boMoveLwConveyorDown;
	                #internal.panel[#PB_Configuration.itOutCmdPbID].boMoving := #EQExitConvR."to".boMoveConveyorFwd OR #EQExitConvR."to".boMoveLwConveyorFwd;
	                #internal.panel[#PB_Configuration.itLockCmdPbID].boMoving := #EQExitConvR."to".boMoveBlockIns OR #EQExitConvR."to".boMoveLwBlockIns;
	                #internal.panel[#PB_Configuration.itUnlockCmdPbID].boMoving := #EQExitConvR."to".boMoveBlockRel OR #EQExitConvR."to".boMoveLwBlockRel;

	                #internal.panel[#PB_Configuration.itUpCmdPbID].boEnable := #EQExitConvL."to".boEnaConveyorUp OR #EQExitConvR."to".boEnaLwConveyorUp OR #internal.panel[#PB_Configuration.itInCmdPbID].boOnPos OR #internal.panel[#PB_Configuration.itInCmdPbID].boMoving;
	                #internal.panel[#PB_Configuration.itDownCmdPbID].boEnable := #EQExitConvL."to".boEnaConveyorDown OR #EQExitConvR."to".boEnaLwConveyorDown OR #internal.panel[#PB_Configuration.itInCmdPbID].boOnPos OR #internal.panel[#PB_Configuration.itInCmdPbID].boMoving;
	                #internal.panel[#PB_Configuration.itOutCmdPbID].boEnable := #EQExitConvL."to".boEnaConveyorFwd OR #EQExitConvR."to".boEnaLwConveyorFwd OR #internal.panel[#PB_Configuration.itInCmdPbID].boOnPos OR #internal.panel[#PB_Configuration.itInCmdPbID].boMoving;
	                #internal.panel[#PB_Configuration.itLockCmdPbID].boEnable := #EQExitConvL."to".boEnaBlockIns OR #EQExitConvR."to".boEnaLwBlockIns OR #internal.panel[#PB_Configuration.itInCmdPbID].boOnPos OR #internal.panel[#PB_Configuration.itInCmdPbID].boMoving;
	                #internal.panel[#PB_Configuration.itUnlockCmdPbID].boEnable := #EQExitConvL."to".boEnaBlockRel OR #EQExitConvR."to".boEnaLwBlockRel OR #internal.panel[#PB_Configuration.itInCmdPbID].boOnPos OR #internal.panel[#PB_Configuration.itInCmdPbID].boMoving;
	            END_IF;

	        END_IF;
	    END_REGION

	END_REGION

	//=======================================================================================================================================
	//            PRODUCTION PROGRAM AUTO
	//=======================================================================================================================================
	REGION PRODUCTION PROGRAM AUTO
	   REGION LEFT
	        IF #internal.boAutoSelOnPressL THEN
	            #internal.panel[#PB_Configuration.itLeftSelPbID].boAborted := #EQgtsL."to".boStatusAbortedEQ OR #EQloaderL."to".boStatusAbortedEQ OR #EQcenterMechL."to".boStatusAbortedEQ OR #EQintHeatL."to".boStatusAbortedEQ OR
	            #EQpressL."to".boStatusAbortedEQ OR #EQextHeatL."to".boStatusAbortedEQ OR #EQunloaderL."to".boStatusAbortedEQ OR #EQExitConvL."to".boStatusAbortedEQ;
	            #internal.panel[#PB_Configuration.itLeftSelPbID].boHeld := #EQgtsL."to".boStatusHeldEQ OR #EQloaderL."to".boStatusHeldEQ OR #EQcenterMechL."to".boStatusHeldEQ OR #EQintHeatL."to".boStatusHeldEQ OR #EQpressL."to".boStatusHeldEQ OR
	            #EQextHeatL."to".boStatusHeldEQ OR #EQunloaderL."to".boStatusHeldEQ OR #EQExitConvL."to".boStatusHeldEQ OR #unitL."to".boMoldDisabled OR #unitL."to".boLoadDisabled;
	            IF #internal.panel[#PB_Configuration.itLeftSelPbID].boSelect THEN
	                REGION LOADER & MGTS & UNIT
	                    #internal.panel[#PB_Configuration.itLoaderPbID].boEnable := TRUE;
	                    #internal.panel[#PB_Configuration.itGTSPbID].boEnable := TRUE;

	                    IF NOT #internal.panel[#PB_Configuration.itRightSelPbID].boSelect THEN
	                        // Modules fault & warning
	                        #internal.panel[#PB_Configuration.itGTSPbID].boAborted := #EQgtsL."to".boStatusAbortedEQ;
	                        #internal.panel[#PB_Configuration.itGTSPbID].boHeld := #EQgtsL."to".boStatusHeldEQ;
	                        #internal.panel[#PB_Configuration.itLoaderPbID].boAborted := #EQloaderL."to".boStatusAbortedEQ;
	                        #internal.panel[#PB_Configuration.itLoaderPbID].boHeld := #EQloaderL."to".boStatusHeldEQ OR #unitL."to".boLoadDisabled;
	                    END_IF;

	                    // MGTS: automatic command
	                    IF #internal.panel[#PB_Configuration.itGTSPbID].boSelect THEN
	                        #internal.panel[#PB_Configuration.itOnOffSelPbID].boEnable := TRUE;
	                    END_IF;

	                    // Loaders: automatic command
	                    IF #internal.panel[#PB_Configuration.itLoaderPbID].boSelect THEN
	                        #internal.panel[#PB_Configuration.itOnOffSelPbID].boEnable := TRUE;
	                        // Protection for wrong disable timer
	                        #internal.disableFilterLeft(IN := #internal.panel[#PB_Configuration.itOnOffSelPbID].boCmdOn AND NOT #internal.boDisableEQLmem,
	                                                   PT := T#2s,
	                                                   Q => #internal.boDisableEQLmem);

	                        IF #internal.boDisableEQLmem AND #internal.panel[#PB_Configuration.itLeftSelPbID].boSelect THEN
	                            #unitL.from.boLoadDisableReq := TRUE;
	                        END_IF;
	                    END_IF;

	                    // Unit procedure commands: pick-up
	                    #internal.panel[#PB_Configuration.itUnitPbID].boEnable := #internal.panel[#PB_Configuration.itUnitPbID].boAborted OR #internal.panel[#PB_Configuration.itUnitPbID].boHeld;
	                    #internal.panel[#PB_Configuration.itPickupPbID].boEnable := #unitL."to".boEnaPickUp OR #internal.panel[#PB_Configuration.itPickupPbID].boAborted; //AND internal.panel[itLeftSelPbID].boSelect;

	                    // Modules fault & warning
	                    #internal.panel[#PB_Configuration.itUnitPbID].boAborted := #unitL."to".boStatusAbortedEQ;
	                    #internal.panel[#PB_Configuration.itPickupPbID].boAborted := #unitL."to".boRescueTireOccured;
	                    #internal.panel[#PB_Configuration.itUnitPbID].boHeld := #unitL."to".boStatusHeldEQ;

	                    // Pick-up command
	                    IF #internal.panel[#PB_Configuration.itPickupPbID].boSelect THEN
	                        #internal.panel[#PB_Configuration.itOnOffSelPbID].boEnable := TRUE;
	                        #internal.panel[#PB_Configuration.itLeftSelPbID].boSelect := #unitL."to".boEnaPickUp AND NOT #unitL."to".boLoadDisabled;
	                        #unitL.from.boPickUpCmd := #internal.panel[#PB_Configuration.itOnOffSelPbID].boCmdRE AND #internal.panel[#PB_Configuration.itLeftSelPbID].boSelect AND #unitL."to".boEnaPickUp AND NOT #unitL."to".boLoadDisabled;
	                    END_IF;

	                END_REGION

	                REGION PRESSES
	                    #internal.panel[#PB_Configuration.itPressPbID].boEnable := TRUE;

	                    IF NOT #internal.panel[#PB_Configuration.itRightSelPbID].boSelect THEN
	                        // Modules fault & warning
	                        #internal.panel[#PB_Configuration.itPressPbID].boAborted := #EQpressL."to".boStatusAbortedEQ;
	                        #internal.panel[#PB_Configuration.itPressPbID].boHeld := #EQpressL."to".boStatusHeldEQ OR #unitL."to".boMoldDisabled;
	                    END_IF;

	                    // Press: automatic commands
	                    IF #internal.panel[#PB_Configuration.itPressPbID].boSelect THEN
	                        #internal.panel[#PB_Configuration.itOnOffSelPbID].boEnable := TRUE;
	                        IF #internal.panel[#PB_Configuration.itOnOffSelPbID].boCmdRE AND FALSE THEN
	                            #unitL.from.boMoldDisableReq := TRUE;
	                        END_IF;
	                    END_IF;
	                END_REGION

	                REGION CENTER-MECH
	                    #internal.panel[#PB_Configuration.itTopRingPbID].boEnable := TRUE;// internal.panel[itTopRingPbID].boAborted OR internal.panel[itTopRingPbID].boHeld;
	                    #internal.panel[#PB_Configuration.itBotRingPbID].boEnable := TRUE;// internal.panel[itBotRingPbID].boAborted OR internal.panel[itBotRingPbID].boHeld;
	                    #internal.panel[#PB_Configuration.itBeadRingPbID].boEnable := TRUE;// internal.panel[itBeadRingPbID].boAborted OR internal.panel[itBeadRingPbID].boHeld;

	                    IF NOT #internal.panel[#PB_Configuration.itRightSelPbID].boSelect THEN
	                        // Modules fault & warning
	                        #internal.panel[#PB_Configuration.itTopRingPbID].boAborted := #EQcenterMechL."to".boStatusAbortedEQ OR #EQcenterMechL."to".boStatusAbortedTCRing;
	                        #internal.panel[#PB_Configuration.itTopRingPbID].boHeld := #EQcenterMechL."to".boStatusHeldEQ OR #EQcenterMechL."to".boStatusHeldTCRing;
	                        #internal.panel[#PB_Configuration.itBotRingPbID].boAborted := #EQcenterMechL."to".boStatusAbortedEQ OR #EQcenterMechL."to".boStatusAbortedBCRing;
	                        #internal.panel[#PB_Configuration.itBotRingPbID].boHeld := #EQcenterMechL."to".boStatusHeldEQ OR #EQcenterMechL."to".boStatusHeldBCRing;
	                        #internal.panel[#PB_Configuration.itBeadRingPbID].boAborted := #EQcenterMechL."to".boStatusAbortedEQ OR #EQcenterMechL."to".boStatusAbortedBeadRing;
	                        #internal.panel[#PB_Configuration.itBeadRingPbID].boHeld := #EQcenterMechL."to".boStatusHeldEQ OR #EQcenterMechL."to".boStatusHeldBeadRing;
	                    END_IF;
	                    // Top Ring: automatic commands
	                    IF #internal.panel[#PB_Configuration.itTopRingPbID].boSelect THEN
	                        #internal.panel[#PB_Configuration.itOnOffSelPbID].boEnable := TRUE;
	                    END_IF;
	                    // Bottom Ring: automatic commands
	                    IF #internal.panel[#PB_Configuration.itBotRingPbID].boSelect THEN
	                        #internal.panel[#PB_Configuration.itOnOffSelPbID].boEnable := TRUE;
	                    END_IF;
	                    // Bead Ring: automatic commands
	                    IF #internal.panel[#PB_Configuration.itBeadRingPbID].boSelect THEN
	                        #internal.panel[#PB_Configuration.itOnOffSelPbID].boEnable := TRUE;
	                    END_IF;
	                END_REGION

	                REGION UNLOADER & COOLING CONVEYORS
	                #internal.panel[#PB_Configuration.itUnloaderPbID].boEnable := TRUE;
	                #internal.panel[#PB_Configuration.itUnloaderPCIPbID].boEnable := TRUE;
	                #internal.panel[#PB_Configuration.itExitConvPbId].boEnable := TRUE;

	                IF NOT #internal.panel[#PB_Configuration.itRightSelPbID].boSelect THEN
	                    // Modules fault & warning
	                    #internal.panel[#PB_Configuration.itUnloaderPbID].boAborted := #EQunloaderL."to".boStatusAbortedEQ;
	                    #internal.panel[#PB_Configuration.itUnloaderPbID].boHeld := #EQunloaderL."to".boStatusHeldEQ;
	                    #internal.panel[#PB_Configuration.itUnloaderPCIPbID].boAborted := #EQunloaderL."to".boStatusAbortedEQ;
	                    #internal.panel[#PB_Configuration.itUnloaderPCIPbID].boHeld := #EQunloaderL."to".boStatusHeldEQ;
	                    #internal.panel[#PB_Configuration.itExitConvPbId].boAborted := #EQExitConvL."to".boStatusAbortedEQ;
	                    #internal.panel[#PB_Configuration.itExitConvPbId].boHeld := #EQExitConvL."to".boStatusHeldEQ;
	                END_IF;
	                // Unloader: automatic commands
	                IF #internal.panel[#PB_Configuration.itUnloaderPbID].boSelect OR #internal.panel[#PB_Configuration.itUnloaderPCIPbID].boSelect THEN
	                    #internal.panel[#PB_Configuration.itOnOffSelPbID].boEnable := TRUE;
	                    IF #internal.panel[#PB_Configuration.itOnOffSelPbID].boCmdRE THEN
	                        #unitL.from.boUnloadDisableReq := TRUE;
	                    END_IF;
	                END_IF;

	                // Cooling conveyors: automatic commands
	                IF #internal.panel[#PB_Configuration.itExitConvPbId].boSelect THEN
	                    #internal.panel[#PB_Configuration.itOnOffSelPbID].boEnable := TRUE;
	                END_IF;
	            END_REGION
	        END_IF;
	        END_IF;
	    END_REGION

	    REGION RIGHT
	    IF #internal.boAutoSelOnPressR THEN
	        #internal.panel[#PB_Configuration.itRightSelPbID].boAborted := #EQgtsR."to".boStatusAbortedEQ OR #EQloaderR."to".boStatusAbortedEQ OR #EQcenterMechR."to".boStatusAbortedEQ OR #EQintHeatR."to".boStatusAbortedEQ OR
	        #EQpressR."to".boStatusAbortedEQ OR #EQextHeatR."to".boStatusAbortedEQ OR #EQunloaderR."to".boStatusAbortedEQ OR #EQExitConvR."to".boStatusAbortedEQ;
	        #internal.panel[#PB_Configuration.itRightSelPbID].boHeld := #EQgtsR."to".boStatusHeldEQ OR #EQloaderR."to".boStatusHeldEQ OR #EQcenterMechR."to".boStatusHeldEQ OR #EQintHeatR."to".boStatusHeldEQ OR #EQpressR."to".boStatusHeldEQ OR
	        #EQextHeatR."to".boStatusHeldEQ OR #EQunloaderR."to".boStatusHeldEQ OR #EQExitConvR."to".boStatusHeldEQ OR #unitR."to".boMoldDisabled OR #unitR."to".boLoadDisabled;


	        IF #internal.panel[#PB_Configuration.itRightSelPbID].boSelect THEN
	            REGION LOADER & MGTS & UNIT
	                #internal.panel[#PB_Configuration.itLoaderPbID].boEnable := TRUE;
	                #internal.panel[#PB_Configuration.itGTSPbID].boEnable := TRUE;

	                IF NOT #internal.panel[#PB_Configuration.itLeftSelPbID].boSelect THEN
	                    // Modules fault & warning
	                    #internal.panel[#PB_Configuration.itGTSPbID].boAborted := #EQgtsR."to".boStatusAbortedEQ;
	                    #internal.panel[#PB_Configuration.itGTSPbID].boHeld := #EQgtsR."to".boStatusHeldEQ;
	                    #internal.panel[#PB_Configuration.itLoaderPbID].boAborted := #EQloaderR."to".boStatusAbortedEQ;
	                    #internal.panel[#PB_Configuration.itLoaderPbID].boHeld := #EQloaderR."to".boStatusHeldEQ OR #unitR."to".boLoadDisabled;
	                END_IF;

	                // MGTS: automatic command
	                IF #internal.panel[#PB_Configuration.itGTSPbID].boSelect THEN
	                    #internal.panel[#PB_Configuration.itOnOffSelPbID].boEnable := TRUE;
	                END_IF;

	                // Loaders: automatic command
	                IF #internal.panel[#PB_Configuration.itLoaderPbID].boSelect THEN
	                    #internal.panel[#PB_Configuration.itOnOffSelPbID].boEnable := TRUE;

	                    // Protection for wrong disable timer
	                    #internal.disableFilterRight(IN := #internal.panel[#PB_Configuration.itOnOffSelPbID].boCmdOn AND NOT #internal.boDisableEQRmem,
	                                                 PT := T#2s,
	                                                 Q => #internal.boDisableEQRmem);

	                    IF #internal.boDisableEQRmem AND #internal.panel[#PB_Configuration.itRightSelPbID].boSelect THEN
	                        #unitR.from.boLoadDisableReq := TRUE;
	                    END_IF;
	                END_IF;

	                // Unit procedure commands: pick-up
	                #internal.panel[#PB_Configuration.itUnitPbID].boEnable := #internal.panel[#PB_Configuration.itUnitPbID].boAborted OR #internal.panel[#PB_Configuration.itUnitPbID].boHeld;
	                #internal.panel[#PB_Configuration.itPickupPbID].boEnable := #unitR."to".boEnaPickUp OR #internal.panel[#PB_Configuration.itPickupPbID].boAborted; //AND internal.panel[itRightSelPbID].boSelect;

	                // Modules fault & warning
	                #internal.panel[#PB_Configuration.itUnitPbID].boAborted := #unitR."to".boStatusAbortedEQ;
	                #internal.panel[#PB_Configuration.itPickupPbID].boAborted := #unitR."to".boRescueTireOccured;
	                #internal.panel[#PB_Configuration.itUnitPbID].boHeld := #unitR."to".boStatusHeldEQ;

	                // Pick-up command
	                IF #internal.panel[#PB_Configuration.itPickupPbID].boSelect THEN
	                    #internal.panel[#PB_Configuration.itOnOffSelPbID].boEnable := TRUE;
	                    #internal.panel[#PB_Configuration.itRightSelPbID].boSelect := #unitR."to".boEnaPickUp AND NOT #unitR."to".boLoadDisabled;
	                    #unitR.from.boPickUpCmd := #internal.panel[#PB_Configuration.itOnOffSelPbID].boCmdRE AND #internal.panel[#PB_Configuration.itRightSelPbID].boSelect AND #unitR."to".boEnaPickUp AND NOT #unitR."to".boLoadDisabled;
	                END_IF;
	            END_REGION
	            REGION PRESSES
	                #internal.panel[#PB_Configuration.itPressPbID].boEnable := TRUE;

	                IF NOT #internal.panel[#PB_Configuration.itLeftSelPbID].boSelect THEN
	                    // Modules fault & warning
	                    #internal.panel[#PB_Configuration.itPressPbID].boAborted := #EQpressR."to".boStatusAbortedEQ;
	                    #internal.panel[#PB_Configuration.itPressPbID].boHeld := #EQpressR."to".boStatusHeldEQ OR #unitR."to".boMoldDisabled;
	                END_IF;

	                // Press: automatic commands
	                IF #internal.panel[#PB_Configuration.itPressPbID].boSelect THEN
	                    #internal.panel[#PB_Configuration.itOnOffSelPbID].boEnable := TRUE;
	                    IF #internal.panel[#PB_Configuration.itOnOffSelPbID].boCmdRE AND FALSE THEN
	                        #unitR.from.boMoldDisableReq := TRUE;
	                    END_IF;
	                END_IF;
	            END_REGION
	            REGION CENTER-MECH
	                #internal.panel[#PB_Configuration.itTopRingPbID].boEnable := TRUE;// internal.panel[itTopRingPbID].boAborted OR internal.panel[itTopRingPbID].boHeld;
	                #internal.panel[#PB_Configuration.itBotRingPbID].boEnable := TRUE;// internal.panel[itBotRingPbID].boAborted OR internal.panel[itBotRingPbID].boHeld;
	                #internal.panel[#PB_Configuration.itBeadRingPbID].boEnable := TRUE;// internal.panel[itBeadRingPbID].boAborted OR internal.panel[itBeadRingPbID].boHeld;

	                IF NOT #internal.panel[#PB_Configuration.itLeftSelPbID].boSelect THEN
	                    // Modules fault & warning
	                    #internal.panel[#PB_Configuration.itTopRingPbID].boAborted := #EQcenterMechR."to".boStatusAbortedEQ OR #EQcenterMechR."to".boStatusAbortedTCRing;
	                    #internal.panel[#PB_Configuration.itTopRingPbID].boHeld := #EQcenterMechR."to".boStatusHeldEQ OR #EQcenterMechR."to".boStatusHeldTCRing;
	                    #internal.panel[#PB_Configuration.itBotRingPbID].boAborted := #EQcenterMechR."to".boStatusAbortedEQ OR #EQcenterMechR."to".boStatusAbortedBCRing;
	                    #internal.panel[#PB_Configuration.itBotRingPbID].boHeld := #EQcenterMechR."to".boStatusHeldEQ OR #EQcenterMechR."to".boStatusHeldBCRing;
	                    #internal.panel[#PB_Configuration.itBeadRingPbID].boAborted := #EQcenterMechR."to".boStatusAbortedEQ OR #EQcenterMechR."to".boStatusAbortedBeadRing;
	                    #internal.panel[#PB_Configuration.itBeadRingPbID].boHeld := #EQcenterMechR."to".boStatusHeldEQ OR #EQcenterMechR."to".boStatusHeldBeadRing;
	                END_IF;

	                // Top Ring: automatic commands
	                IF #internal.panel[#PB_Configuration.itTopRingPbID].boSelect THEN
	                    #internal.panel[#PB_Configuration.itOnOffSelPbID].boEnable := TRUE;
	                END_IF;
	                // Bottom Ring: automatic commands
	                IF #internal.panel[#PB_Configuration.itBotRingPbID].boSelect THEN
	                    #internal.panel[#PB_Configuration.itOnOffSelPbID].boEnable := TRUE;
	                END_IF;
	                // Bead Ring: automatic commands
	                IF #internal.panel[#PB_Configuration.itBeadRingPbID].boSelect THEN
	                    #internal.panel[#PB_Configuration.itOnOffSelPbID].boEnable := TRUE;
	                END_IF;
	            END_REGION
	            REGION UNLOADER & COOLING CONVEYORS
	                #internal.panel[#PB_Configuration.itUnloaderPbID].boEnable := TRUE;
	                #internal.panel[#PB_Configuration.itUnloaderPCIPbID].boEnable := TRUE;
	                #internal.panel[#PB_Configuration.itExitConvPbId].boEnable := TRUE;

	                IF NOT #internal.panel[#PB_Configuration.itLeftSelPbID].boSelect THEN
	                    // Modules fault & warning
	                    #internal.panel[#PB_Configuration.itUnloaderPbID].boAborted := #EQunloaderR."to".boStatusAbortedEQ;
	                    #internal.panel[#PB_Configuration.itUnloaderPbID].boHeld := #EQunloaderR."to".boStatusHeldEQ;
	                    #internal.panel[#PB_Configuration.itUnloaderPCIPbID].boAborted := #EQunloaderR."to".boStatusAbortedEQ;
	                    #internal.panel[#PB_Configuration.itUnloaderPCIPbID].boHeld := #EQunloaderR."to".boStatusHeldEQ;
	                    #internal.panel[#PB_Configuration.itExitConvPbId].boAborted := #EQExitConvR."to".boStatusAbortedEQ;
	                    #internal.panel[#PB_Configuration.itExitConvPbId].boHeld := #EQExitConvR."to".boStatusHeldEQ;
	                END_IF;

	                // Unloader: automatic commands
	                IF #internal.panel[#PB_Configuration.itUnloaderPbID].boSelect OR #internal.panel[#PB_Configuration.itUnloaderPCIPbID].boSelect THEN
	                    #internal.panel[#PB_Configuration.itOnOffSelPbID].boEnable := TRUE;
	                    IF #internal.panel[#PB_Configuration.itOnOffSelPbID].boCmdRE THEN
	                        #unitR.from.boUnloadDisableReq := TRUE;
	                    END_IF;
	                END_IF;

	                IF #internal.panel[#PB_Configuration.itExitConvPbId].boSelect THEN
	                    #internal.panel[#PB_Configuration.itOnOffSelPbID].boEnable := TRUE;
	                END_IF;
	            END_REGION
	        END_IF;
	    END_IF;
	END_REGION

	    REGION HEATING (INTERNAL & EXTERNAL)
	    IF #internal.boAutoSelOnHeatingL THEN
	        #internal.panel[#PB_Configuration.itShapingPbID].boEnable := TRUE;
	        #internal.panel[#PB_Configuration.itExtHeatingPbID].boEnable := TRUE;

	        IF NOT #internal.panel[#PB_Configuration.itRightSelPbID].boSelect THEN
	            // Unit curing active
	            #internal.panel[#PB_Configuration.itShapingPbID].boMoving := #EQintHeatL."to".boCuringActive;

	            // Unit procedure commands: gym
	            #internal.panel[#PB_Configuration.itGymPbID].boEnable := #unitL."to".boEnaGym OR #unitL."to".boGymActivated;
	            #internal.panel[#PB_Configuration.itGymPbID].boHeld := #unitL."to".boGymActivated AND NOT #internal.panel[#PB_Configuration.itGymPbID].boSelect;
	            #internal.panel[#PB_Configuration.itExtHeatingPbID].boHeld := NOT #unitL."to".boMoldPrewarmDone AND NOT #unitL."to".boMoldDisabled;

	            // External heating pre-warm done
	            #internal.panel[#PB_Configuration.itLeftSelPbID].boHeld := NOT #unitL."to".boMoldPrewarmDone AND NOT #unitL."to".boMoldDisabled;
	        END_IF;

	        IF #internal.panel[#PB_Configuration.itGymPbID].boSelect THEN
	            #internal.panel[#PB_Configuration.itOnOffSelPbID].boEnable := TRUE;
	            #unitL.from.boGymCmd := #internal.panel[#PB_Configuration.itLeftSelPbID].boSelect AND #internal.panel[#PB_Configuration.itOnOffSelPbID].boCmdRE;
	        END_IF;

	    END_IF;

	    IF #internal.boAutoSelOnHeatingR THEN
	        #internal.panel[#PB_Configuration.itShapingPbID].boEnable := TRUE;
	        #internal.panel[#PB_Configuration.itExtHeatingPbID].boEnable := TRUE;

	        IF NOT #internal.panel[#PB_Configuration.itLeftSelPbID].boSelect THEN
	            // Unit curing active
	            #internal.panel[#PB_Configuration.itShapingPbID].boMoving := #EQintHeatR."to".boCuringActive;

	            // Unit procedure commands: gym
	            #internal.panel[#PB_Configuration.itGymPbID].boEnable := #unitR."to".boEnaGym OR #unitR."to".boGymActivated;
	            #internal.panel[#PB_Configuration.itGymPbID].boHeld := #unitR."to".boGymActivated AND NOT #internal.panel[#PB_Configuration.itGymPbID].boSelect;
	            #internal.panel[#PB_Configuration.itExtHeatingPbID].boHeld := NOT #unitR."to".boMoldPrewarmDone AND NOT #unitR."to".boMoldDisabled;

	            // External heating pre-warm done
	            #internal.panel[#PB_Configuration.itRightSelPbID].boHeld := NOT #unitR."to".boMoldPrewarmDone AND NOT #unitR."to".boMoldDisabled;
	        END_IF;

	        IF #internal.panel[#PB_Configuration.itGymPbID].boSelect THEN
	            #internal.panel[#PB_Configuration.itOnOffSelPbID].boEnable := TRUE;
	            #unitR.from.boGymCmd := #internal.panel[#PB_Configuration.itRightSelPbID].boSelect AND #internal.panel[#PB_Configuration.itOnOffSelPbID].boCmdRE;
	        END_IF;
	    END_IF;

	    IF #internal.boAutoSelOnHeatingL AND #internal.panel[#PB_Configuration.itLeftSelPbID].boSelect AND
	        #internal.boAutoSelOnHeatingR AND #internal.panel[#PB_Configuration.itRightSelPbID].boSelect THEN
	        // Unit curing active
	        #internal.panel[#PB_Configuration.itShapingPbID].boMoving := #EQintHeatL."to".boCuringActive OR #EQintHeatR."to".boCuringActive;
	        // Unit procedure commands: gym
	        #internal.panel[#PB_Configuration.itGymPbID].boEnable := #unitL."to".boEnaGym OR #unitL."to".boGymActivated OR #unitR."to".boEnaGym OR #unitR."to".boGymActivated;
	        #internal.panel[#PB_Configuration.itGymPbID].boHeld := (#unitL."to".boGymActivated OR #unitR."to".boGymActivated) AND NOT #internal.panel[#PB_Configuration.itGymPbID].boSelect;
	        #internal.panel[#PB_Configuration.itExtHeatingPbID].boHeld := (NOT #unitL."to".boMoldPrewarmDone AND NOT #unitL."to".boMoldDisabled) OR (NOT #unitR."to".boMoldPrewarmDone AND NOT #unitR."to".boMoldDisabled);

	        // External heating pre-warm done
	        #internal.panel[#PB_Configuration.itLeftSelPbID].boHeld := NOT #unitL."to".boMoldPrewarmDone AND NOT #unitL."to".boMoldDisabled;
	        #internal.panel[#PB_Configuration.itRightSelPbID].boHeld := NOT #unitR."to".boMoldPrewarmDone AND NOT #unitR."to".boMoldDisabled;
	    END_IF;

	    //COMMON PART WHEN WE ARE ON BOTH SIDE IN AUTOMATIC AND BOTH SELECTED TO SHOW ALARM ON EACH SIDE PUSHBUTTON
	    //  IF internal.boAutoSelOnPressL AND internal.boAutoSelOnPressR THEN
	    //      internal.panel[itLeftSelPbID].boHeld := EQgtsL."to".boStatusHeldEQ OR EQloaderL."to".boStatusHeldEQ OR EQcenterMechL."to".boStatusHeldEQ OR EQintHeatL."to".boStatusHeldEQ OR EQpressL."to".boStatusHeldEQ OR
	    //                                              EQextHeatL."to".boStatusHeldEQ OR EQunloaderL."to".boStatusHeldEQ OR EQExitConvL."to".boStatusHeldEQ OR unitL."to".boMoldDisabled OR unitL."to".boLoadDisabled;
	    //      internal.panel[itRightSelPbID].boHeld := EQgtsR."to".boStatusHeldEQ OR EQloaderR."to".boStatusHeldEQ OR EQcenterMechR."to".boStatusHeldEQ OR EQintHeatR."to".boStatusHeldEQ OR EQpressR."to".boStatusHeldEQ OR
	    //                                               EQextHeatR."to".boStatusHeldEQ OR EQunloaderR."to".boStatusHeldEQ OR EQExitConvR."to".boStatusHeldEQ OR unitR."to".boMoldDisabled OR unitR."to".boLoadDisabled;
	    //  END_IF;
	END_REGION

	END_REGION

	//=======================================================================================================================================
	//            SETUP PROGRAM
	//=======================================================================================================================================
	REGION SETUP PROGRAM
	    #internal.boSetupProcActiveL := FALSE;
	    IF (#internal.boSetupSelOnHeatingL AND #internal.boSetupSelOnPressL) AND #internal.panel[#PB_Configuration.itLeftSelPbID].boSelect THEN

	        // Equipments free manual commands enable
	        #internal.boSetupProcActiveL := #unitL."to".boSetupProcActive;

	        IF NOT #unitL."to".boSetupFreeManualActive THEN
	            // Start bladder change from panel
	            //#internal.panel[#PB_Configuration.itGymPbID].boEnable := #unitL."to".boSetupBladderChangeEna;
	            //#internal.panel[#PB_Configuration.itOnOffSelPbID].boEnable := #unitL."to".boSetupBladderChangeEna;
	            #unitL.from.boSetupBladderChangeReq := #internal.panel[#PB_Configuration.itGymPbID].boSelect AND #internal.panel[#PB_Configuration.itOnOffSelPbID].boCmdOn AND #unitL."to".boSetupBladderChangeEna;

	            // Start mold change from panel
	            //#internal.panel[#PB_Configuration.itSegmentsPbID].boEnable := #unitL."to".boSetupMoldChangeEna;
	            //#internal.panel[#PB_Configuration.itOnOffSelPbID].boEnable := #unitL."to".boSetupMoldChangeEna;
	            #unitL.from.boSetupMoldChangeReq := #internal.panel[#PB_Configuration.itSegmentsPbID].boSelect AND #internal.panel[#PB_Configuration.itOnOffSelPbID].boCmdOn AND #unitL."to".boSetupMoldChangeEna;
	        END_IF;

	        // Moves to next step or to completation of procedure
	        IF #internal.panel[#PB_Configuration.itLeftSelPbID].boSelect THEN
	            #internal.panel[#PB_Configuration.itNextCmdPbID].boEnable := #unitL."to".boSetupProcActive AND #unitL."to".boSetupProcEnaNextStep;
	            #unitL.from.boSetupProcNextStep := #internal.panel[#PB_Configuration.itNextCmdPbID].boCmdRE;
	        END_IF;
	    END_IF;

	    #internal.boSetupProcActiveR := FALSE;
	    IF (#internal.boSetupSelOnHeatingR AND #internal.boSetupSelOnPressR) AND #internal.panel[#PB_Configuration.itRightSelPbID].boSelect THEN

	        // Equipments free manual commands enable
	        #internal.boSetupProcActiveR := #unitR."to".boSetupProcActive;
	        IF NOT #unitR."to".boSetupFreeManualActive THEN
	            // Start bladder change from panel
	            //#internal.panel[#PB_Configuration.itGymPbID].boEnable := #unitR."to".boSetupBladderChangeEna;
	            //#internal.panel[#PB_Configuration.itOnOffSelPbID].boEnable := #unitR."to".boSetupBladderChangeEna;
	            #unitR.from.boSetupBladderChangeReq := #internal.panel[#PB_Configuration.itGymPbID].boSelect AND #internal.panel[#PB_Configuration.itOnOffSelPbID].boCmdOn AND #unitR."to".boSetupBladderChangeEna;

	            // Start mold change from panel
	            //#internal.panel[#PB_Configuration.itSegmentsPbID].boEnable := #unitL."to".boSetupMoldChangeEna;
	            //#internal.panel[#PB_Configuration.itOnOffSelPbID].boEnable := #unitL."to".boSetupMoldChangeEna;
	            #unitR.from.boSetupMoldChangeReq := #internal.panel[#PB_Configuration.itSegmentsPbID].boSelect AND #internal.panel[#PB_Configuration.itOnOffSelPbID].boCmdOn AND #unitR."to".boSetupMoldChangeEna;
	        END_IF;

	        // Moves to next step or to completation of procedure
	        IF #internal.panel[#PB_Configuration.itRightSelPbID].boSelect THEN
	            #internal.panel[#PB_Configuration.itNextCmdPbID].boEnable := #unitR."to".boSetupProcActive AND #unitR."to".boSetupProcEnaNextStep;
	            #unitR.from.boSetupProcNextStep := #internal.panel[#PB_Configuration.itNextCmdPbID].boCmdRE;
	        END_IF;
	    END_IF;
	END_REGION

	REGION HPU
	    // Enable push-buttons
	    #internal.panel[#PB_Configuration.itHPUPbID].boEnable := TRUE;

	    // Modules fault & warning
	    #internal.panel[#PB_Configuration.itHPUPbID].boAborted := #EQhpu."to".boStatusAbortedEQ;
	    #internal.panel[#PB_Configuration.itHPUPbID].boHeld := #EQhpu."to".boStatusHeldEQ;

	    IF #internal.panel[#PB_Configuration.itHPUPbID].boSelect THEN
	        #internal.panel[#PB_Configuration.itLeftSelPbID].boAborted := #EQhpu."to".boStatusAbortedEQ;
	        #internal.panel[#PB_Configuration.itRightSelPbID].boAborted := #EQhpu."to".boStatusAbortedEQ;
	        #internal.panel[#PB_Configuration.itLeftSelPbID].boHeld := #EQhpu."to".boStatusHeldEQ;
	        #internal.panel[#PB_Configuration.itRightSelPbID].boHeld := #EQhpu."to".boStatusHeldEQ;

	        IF #internal.panel[#PB_Configuration.itHPUPbID].boSelect AND NOT #internal.boHPU_Selected THEN
	            #internal.panel[#PB_Configuration.itLeftSelPbID].boSelect := TRUE;
	            #internal.panel[#PB_Configuration.itRightSelPbID].boSelect := TRUE;
	        END_IF;

	        #internal.panel[#PB_Configuration.itOnOffSelPbID].boOnPos := (#EQhpu."to".boPosPumpRunning AND #internal.panel[#PB_Configuration.itLeftSelPbID].boSelect) AND
	                                                    (#EQhpu."to".boPosPumpRunning AND #internal.panel[#PB_Configuration.itRightSelPbID].boSelect);
	        #internal.panel[#PB_Configuration.itUpCmdPbID].boOnPos := FALSE;//(#EQhpu."to".boPosHPVlvOpen AND #internal.panel[#PB_Configuration.itLeftSelPbID].boSelect) AND
	                                                 //(#EQhpu."to".boPosHPVlvOpen AND #internal.panel[#PB_Configuration.itRightSelPbID].boSelect);
	        #internal.panel[#PB_Configuration.itDownCmdPbID].boOnPos := FALSE;//(#EQhpu."to".boPosLPLeftVlvOpen AND #internal.panel[#PB_Configuration.itLeftSelPbID].boSelect) AND
	                                                   //(#EQhpu."to".boPosLPRightVlvOpen AND #internal.panel[#PB_Configuration.itRightSelPbID].boSelect);

	        #internal.panel[#PB_Configuration.itOnOffSelPbID].boMoving := (#EQhpu."to".boMovePumpRunning AND #internal.panel[#PB_Configuration.itLeftSelPbID].boSelect) OR
	                                                     (#EQhpu."to".boMovePumpRunning AND #internal.panel[#PB_Configuration.itRightSelPbID].boSelect);
	        #internal.panel[#PB_Configuration.itUpCmdPbID].boMoving := FALSE;//(#EQhpu."to".boMoveHPVlvOpen AND #internal.panel[#PB_Configuration.itLeftSelPbID].boSelect) OR
	                                                  //(#EQhpu."to".boMoveHPVlvOpen AND #internal.panel[#PB_Configuration.itRightSelPbID].boSelect);
	        #internal.panel[#PB_Configuration.itDownCmdPbID].boMoving := FALSE;//(#EQhpu."to".boMoveLPLeftVlvOpen AND #internal.panel[#PB_Configuration.itLeftSelPbID].boSelect) OR
	                                                    //(#EQhpu."to".boMoveLPRightVlvOpen AND #internal.panel[#PB_Configuration.itRightSelPbID].boSelect);

	        IF (#internal.boManSelOnPressL AND #internal.boManSelOnPressR) OR (#internal.boSetupSelOnPressL AND #internal.boSetupSelOnPressR) OR
	            (#internal.boSetupProcActiveL AND #internal.boSetupProcActiveR) THEN
	            #internal.panel[#PB_Configuration.itOnOffSelPbID].boEnable := (#EQhpu."to".boEnaPumpRun AND #internal.panel[#PB_Configuration.itLeftSelPbID].boSelect) OR
	                                                         (#EQhpu."to".boEnaPumpRun AND #internal.panel[#PB_Configuration.itRightSelPbID].boSelect);
	            #internal.panel[#PB_Configuration.itUpCmdPbID].boEnable := FALSE;//(#EQhpu."to".boEnaHPVlvOpen AND #internal.panel[#PB_Configuration.itLeftSelPbID].boSelect) OR
	                                                      //(#EQhpu."to".boEnaHPVlvOpen AND #internal.panel[#PB_Configuration.itRightSelPbID].boSelect);
	            #internal.panel[#PB_Configuration.itDownCmdPbID].boEnable := FALSE;//(#EQhpu."to".boEnaLPLeftVlvOpen AND #internal.panel[#PB_Configuration.itLeftSelPbID].boSelect) OR
	                                                        //(#EQhpu."to".boEnaLPRightVlvOpen AND #internal.panel[#PB_Configuration.itRightSelPbID].boSelect);

	            #EQhpu.from.boSelected := #internal.panel[#PB_Configuration.itHPUPbID].boSelect;
	            #EQhpu.from.boLeftSideSelected := #internal.panel[#PB_Configuration.itLeftSelPbID].boSelect;
	            #EQhpu.from.boRightSideSelected := #internal.panel[#PB_Configuration.itRightSelPbID].boSelect;
	            #EQhpu.from.boCmdStartHPU := #internal.panel[#PB_Configuration.itOnOffSelPbID].boCmdOn AND (#internal.panel[#PB_Configuration.itLeftSelPbID].boSelect OR #internal.panel[#PB_Configuration.itRightSelPbID].boSelect);
	            #EQhpu.from.boCmdRequiredOilLPLeft := #internal.panel[#PB_Configuration.itDownCmdPbID].boCmdOn AND #internal.panel[#PB_Configuration.itLeftSelPbID].boSelect;
	            #EQhpu.from.boCmdRequiredOilLPRight := #internal.panel[#PB_Configuration.itDownCmdPbID].boCmdOn AND #internal.panel[#PB_Configuration.itRightSelPbID].boSelect;
	            #EQhpu.from.boCmdRequiredOilHP := #internal.panel[#PB_Configuration.itUpCmdPbID].boCmdOn AND (#internal.panel[#PB_Configuration.itLeftSelPbID].boSelect OR #internal.panel[#PB_Configuration.itRightSelPbID].boSelect);
	        END_IF;
	    END_IF;
	    #internal.boHPU_Selected := #internal.panel[#PB_Configuration.itHPUPbID].boSelect;
	END_REGION

	//=======================================================================================================================================
	//            WRITE OUTPUTS TO KP32F
	//=======================================================================================================================================
	REGION WRITE OUTPUTS TO KP32F
	    // Reset all PBs states
	    IF #boResetPBsStatesTemp THEN
	        FOR #itPushButtonIndexTemp := 0 TO 31 DO
	            #internal.panel[#itPushButtonIndexTemp].boHeld := FALSE;
	            #internal.panel[#itPushButtonIndexTemp].boAborted := FALSE;
	            #internal.panel[#itPushButtonIndexTemp].boMoving := FALSE;
	            #internal.panel[#itPushButtonIndexTemp].boOnPos := FALSE;
	            #internal.panel[#itPushButtonIndexTemp].boInterlock := FALSE;
	            #internal.panel[#itPushButtonIndexTemp].boDisabled := FALSE;
	            IF (#internal.panel[#itPushButtonIndexTemp].itPBType = #PB_COMMAND) THEN
	                #internal.panel[#itPushButtonIndexTemp].boEnable := FALSE;
	                #internal.panel[#itPushButtonIndexTemp].boSelect := FALSE;
	            END_IF;
	        END_FOR;
	    END_IF;

	    // Wrong button pushed timer
	    #internal.disabledTOF(IN := #boWrongPushCmdTemp,
	                          PT := T#1s,
	                          Q => #internal.boWrongPushCmdFilt);

	    // Test lamp
	    #internal.testLampTON(IN := #internal.panel[#PB_Configuration.itLampTestPbID].boCmdOn AND NOT #internal.boChgOfTestLampIndex,
	                          PT := T#1s,
	                          Q => #internal.boChgOfTestLampIndex);
	    IF NOT #internal.panel[#PB_Configuration.itLampTestPbID].boCmdOn THEN
	        #internal.itTestLampIndex := 0;
	    ELSIF (#internal.itTestLampIndex = 0) THEN
	        #internal.itTestLampIndex := 1;
	    ELSIF #internal.boChgOfTestLampIndex THEN
	        #internal.itTestLampIndex := #internal.itTestLampIndex + 1;
	        IF #internal.itTestLampIndex > 5 THEN
	            #internal.itTestLampIndex := 1;
	        END_IF;
	    END_IF;
	    #boTestLampOn := #internal.panel[#PB_Configuration.itLampTestPbID].boCmdOn;
	    // KP32F management of lamps and buttons
	    FOR #itPushButtonIndexTemp := 0 TO 31 DO

	        (*
	        Push buttons lamp management:
	                OUT:   red      green      blue
	        COLOUR:
	            red         1         0         0
	            green       0         1         0
	            blue        0         0         1
	            yellow      1         1         0
	            white       1         1         1
	            OFF         0         0         0
	            OFF         0         1         1
	            OFF         1         0         1

	        Push buttons order in the panel:
	            07  06  05  04  03  02  01  00
	            15  14  13  12  11  10  09  08
	            23  22  21  20  19  18  17  16
	            31  30  29  28  27  26  25  24
	        *)

	        // Lamp colour of button
	        #boRedLampTemp := FALSE;
	        #boGreenLampTemp := FALSE;
	        #boBlueLampTemp := FALSE;
	        #itColourCodeTemp := #COLOUR_NONE;
	        IF #internal.panel[#itPushButtonIndexTemp].boEnable OR #internal.boWrongPushCmdFilt OR #boChgOfModeFiltTemp THEN
	            IF #internal.panel[#itPushButtonIndexTemp].boCmdWrong AND #internal.boWrongPushCmdFilt THEN
	                #itColourCodeTemp := #ColorCode_Configuration.itDisabledColourCode;
	            ELSIF #boChgOfModeFiltTemp THEN
	                IF #internal.panel[#itPushButtonIndexTemp].boSemiAMode THEN
	                    #itColourCodeTemp := #ColorCode_Configuration.itManualColourCode;
	                ELSIF #internal.panel[#itPushButtonIndexTemp].boAutoMode THEN
	                    #itColourCodeTemp := #ColorCode_Configuration.itAutomaticColourCode;
	                END_IF;
	            ELSIF #internal.panel[#itPushButtonIndexTemp].boInterlock THEN
	                #itColourCodeTemp := #ColorCode_Configuration.itInterlockColourCode;
	            ELSIF #internal.panel[#itPushButtonIndexTemp].boAborted THEN
	                IF (#internal.panel[#itPushButtonIndexTemp].itPBType <> #PB_COMMAND) THEN
	                    #itColourCodeTemp := #ColorCode_Configuration.itFaultColourCode;
	                ELSE
	                    #itColourCodeTemp := #ColorCode_Configuration.itCmdPBFaultColourCode;
	                END_IF;
	            ELSIF #internal.panel[#itPushButtonIndexTemp].boHeld THEN
	                IF (#internal.panel[#itPushButtonIndexTemp].itPBType <> #PB_COMMAND) THEN
	                    #itColourCodeTemp := #ColorCode_Configuration.itWarningColourCode;
	                ELSE
	                    #itColourCodeTemp := #ColorCode_Configuration.itCmdPBWarningColourCode;
	                END_IF;
	            ELSIF #internal.panel[#itPushButtonIndexTemp].boMoving THEN
	                IF (#internal.panel[#itPushButtonIndexTemp].itPBType <> #PB_COMMAND) THEN
	                    #itColourCodeTemp := #ColorCode_Configuration.itMoveColourCode;
	                ELSE
	                    #itColourCodeTemp := #ColorCode_Configuration.itCmdPBMoveColourCode;
	                END_IF;
	            ELSIF #internal.panel[#itPushButtonIndexTemp].boOnPos THEN
	                IF (#internal.panel[#itPushButtonIndexTemp].itPBType <> #PB_COMMAND) THEN
	                    #itColourCodeTemp := #ColorCode_Configuration.itOnPosColourCode;
	                ELSE
	                    #itColourCodeTemp := #ColorCode_Configuration.itCmdPBOnPosColourCode;
	                END_IF;
	            ELSIF #internal.panel[#itPushButtonIndexTemp].boSelect THEN
	                IF (#internal.panel[#itPushButtonIndexTemp].itPBType <> #PB_COMMAND) THEN
	                    #itColourCodeTemp := #ColorCode_Configuration.itSelectColourCode;
	                ELSE
	                    #itColourCodeTemp := #ColorCode_Configuration.itCmdPBSelectColourCode;
	                END_IF;
	            ELSE
	                IF (#internal.panel[#itPushButtonIndexTemp].itPBType <> #PB_COMMAND) THEN
	                    #itColourCodeTemp := #ColorCode_Configuration.itEnableColourCode;
	                ELSE
	                    #itColourCodeTemp := #ColorCode_Configuration.itCmdPBEnableColourCode;
	                END_IF;
	            END_IF;
	        END_IF;
	        #internal.simulation[#itPushButtonIndexTemp].itColour := #itColourCodeTemp;
	        CASE #itColourCodeTemp OF
	            #COLOUR_RED:
	                #boRedLampTemp := TRUE;
	                #boGreenLampTemp := FALSE;
	                #boBlueLampTemp := FALSE;
	            #COLOUR_GREEN:
	                #boRedLampTemp := FALSE;
	                #boGreenLampTemp := TRUE;
	                #boBlueLampTemp := FALSE;
	            #COLOUR_BLUE:
	                #boRedLampTemp := FALSE;
	                #boGreenLampTemp := FALSE;
	                #boBlueLampTemp := TRUE;
	            #COLOUR_YELLOW:
	                #boRedLampTemp := TRUE;
	                #boGreenLampTemp := TRUE;
	                #boBlueLampTemp := FALSE;
	            #COLOUR_WHITE:
	                #boRedLampTemp := TRUE;
	                #boGreenLampTemp := TRUE;
	                #boBlueLampTemp := TRUE;
	            #COLOUR_RED_BLINK:
	                #boRedLampTemp := "SYS_Square1000ms";
	                #boGreenLampTemp := FALSE;
	                #boBlueLampTemp := FALSE;
	            #COLOUR_GREEN_BLINK:
	                #boRedLampTemp := FALSE;
	                #boGreenLampTemp := "SYS_Square1000ms";
	                #boBlueLampTemp := FALSE;
	            #COLOUR_BLUE_BLINK:
	                #boRedLampTemp := FALSE;
	                #boGreenLampTemp := FALSE;
	                #boBlueLampTemp := "SYS_Square1000ms";
	            #COLOUR_YELLOW_BLINK:
	                #boRedLampTemp := "SYS_Square1000ms";
	                #boGreenLampTemp := "SYS_Square1000ms";
	                #boBlueLampTemp := FALSE;
	            #COLOUR_WHITE_BLINK:
	                #boRedLampTemp := "SYS_Square1000ms";
	                #boGreenLampTemp := "SYS_Square1000ms";
	                #boBlueLampTemp := "SYS_Square1000ms";
	            #COLOUR_RED_BLINK_FAST:
	                #boRedLampTemp := "SYS_Square500ms";
	                #boGreenLampTemp := FALSE;
	                #boBlueLampTemp := FALSE;
	            #COLOUR_GREEN_BLINK_FAST:
	                #boRedLampTemp := FALSE;
	                #boGreenLampTemp := "SYS_Square500ms";
	                #boBlueLampTemp := FALSE;
	            #COLOUR_BLUE_BLINK_FAST:
	                #boRedLampTemp := FALSE;
	                #boGreenLampTemp := FALSE;
	                #boBlueLampTemp := "SYS_Square500ms";
	            #COLOUR_YELLOW_BLINK_FAST:
	                #boRedLampTemp := "SYS_Square500ms";
	                #boGreenLampTemp := "SYS_Square500ms";
	                #boBlueLampTemp := FALSE;
	            #COLOUR_WHITE_BLINK_FAST:
	                #boRedLampTemp := "SYS_Square500ms";
	                #boGreenLampTemp := "SYS_Square500ms";
	                #boBlueLampTemp := "SYS_Square500ms";
	        END_CASE;
	        IF (#internal.itTestLampIndex <> 0) THEN
	            #boRedLampTemp := (#internal.itTestLampIndex = 1) OR (#internal.itTestLampIndex = 4) OR (#internal.itTestLampIndex = 5);
	            #boGreenLampTemp := (#internal.itTestLampIndex = 2) OR (#internal.itTestLampIndex = 4) OR (#internal.itTestLampIndex = 5);
	            #boBlueLampTemp := (#internal.itTestLampIndex = 3) OR (#internal.itTestLampIndex = 5);
	            IF #boRedLampTemp AND NOT #boGreenLampTemp AND NOT #boBlueLampTemp THEN
	                #internal.simulation[#itPushButtonIndexTemp].itColour := #COLOUR_RED;
	            ELSIF NOT #boRedLampTemp AND #boGreenLampTemp AND NOT #boBlueLampTemp THEN
	                #internal.simulation[#itPushButtonIndexTemp].itColour := #COLOUR_GREEN;
	            ELSIF NOT #boRedLampTemp AND NOT #boGreenLampTemp AND #boBlueLampTemp THEN
	                #internal.simulation[#itPushButtonIndexTemp].itColour := #COLOUR_BLUE;
	            ELSIF #boRedLampTemp AND #boGreenLampTemp AND NOT #boBlueLampTemp THEN
	                #internal.simulation[#itPushButtonIndexTemp].itColour := #COLOUR_YELLOW;
	            ELSIF #boRedLampTemp AND #boGreenLampTemp AND #boBlueLampTemp THEN
	                #internal.simulation[#itPushButtonIndexTemp].itColour := #COLOUR_WHITE;
	            END_IF;
	        END_IF;
	        CASE #itPushButtonIndexTemp OF
	            0:
	                #internal.lamps0_15.red00 := #boRedLampTemp;
	                #internal.lamps0_15.green00 := #boGreenLampTemp;
	                #internal.lamps0_15.blue00 := #boBlueLampTemp;
	            1:
	                #internal.lamps0_15.red01 := #boRedLampTemp;
	                #internal.lamps0_15.green01 := #boGreenLampTemp;
	                #internal.lamps0_15.blue01 := #boBlueLampTemp;
	            2:
	                #internal.lamps0_15.red02 := #boRedLampTemp;
	                #internal.lamps0_15.green02 := #boGreenLampTemp;
	                #internal.lamps0_15.blue02 := #boBlueLampTemp;
	            3:
	                #internal.lamps0_15.red03 := #boRedLampTemp;
	                #internal.lamps0_15.green03 := #boGreenLampTemp;
	                #internal.lamps0_15.blue03 := #boBlueLampTemp;
	            4:
	                #internal.lamps0_15.red04 := #boRedLampTemp;
	                #internal.lamps0_15.green04 := #boGreenLampTemp;
	                #internal.lamps0_15.blue04 := #boBlueLampTemp;
	            5:
	                #internal.lamps0_15.red05 := #boRedLampTemp;
	                #internal.lamps0_15.green05 := #boGreenLampTemp;
	                #internal.lamps0_15.blue05 := #boBlueLampTemp;
	            6:
	                #internal.lamps0_15.red06 := #boRedLampTemp;
	                #internal.lamps0_15.green06 := #boGreenLampTemp;
	                #internal.lamps0_15.blue06 := #boBlueLampTemp;
	            7:
	                #internal.lamps0_15.red07 := #boRedLampTemp;
	                #internal.lamps0_15.green07 := #boGreenLampTemp;
	                #internal.lamps0_15.blue07 := #boBlueLampTemp;
	            8:
	                #internal.lamps0_15.red08 := #boRedLampTemp;
	                #internal.lamps0_15.green08 := #boGreenLampTemp;
	                #internal.lamps0_15.blue08 := #boBlueLampTemp;
	            9:
	                #internal.lamps0_15.red09 := #boRedLampTemp;
	                #internal.lamps0_15.green09 := #boGreenLampTemp;
	                #internal.lamps0_15.blue09 := #boBlueLampTemp;
	            10:
	                #internal.lamps0_15.red10 := #boRedLampTemp;
	                #internal.lamps0_15.green10 := #boGreenLampTemp;
	                #internal.lamps0_15.blue10 := #boBlueLampTemp;
	            11:
	                #internal.lamps0_15.red11 := #boRedLampTemp;
	                #internal.lamps0_15.green11 := #boGreenLampTemp;
	                #internal.lamps0_15.blue11 := #boBlueLampTemp;
	            12:
	                #internal.lamps0_15.red12 := #boRedLampTemp;
	                #internal.lamps0_15.green12 := #boGreenLampTemp;
	                #internal.lamps0_15.blue12 := #boBlueLampTemp;
	            13:
	                #internal.lamps0_15.red13 := #boRedLampTemp;
	                #internal.lamps0_15.green13 := #boGreenLampTemp;
	                #internal.lamps0_15.blue13 := #boBlueLampTemp;
	            14:
	                #internal.lamps0_15.red14 := #boRedLampTemp;
	                #internal.lamps0_15.green14 := #boGreenLampTemp;
	                #internal.lamps0_15.blue14 := #boBlueLampTemp;
	            15:
	                #internal.lamps0_15.red15 := #boRedLampTemp;
	                #internal.lamps0_15.green15 := #boGreenLampTemp;
	                #internal.lamps0_15.blue15 := #boBlueLampTemp;
	            16:
	                #internal.lamps16_31.red16 := #boRedLampTemp;
	                #internal.lamps16_31.green16 := #boGreenLampTemp;
	                #internal.lamps16_31.blue16 := #boBlueLampTemp;
	            17:
	                #internal.lamps16_31.red17 := #boRedLampTemp;
	                #internal.lamps16_31.green17 := #boGreenLampTemp;
	                #internal.lamps16_31.blue17 := #boBlueLampTemp;
	            18:
	                #internal.lamps16_31.red18 := #boRedLampTemp;
	                #internal.lamps16_31.green18 := #boGreenLampTemp;
	                #internal.lamps16_31.blue18 := #boBlueLampTemp;
	            19:
	                #internal.lamps16_31.red19 := #boRedLampTemp;
	                #internal.lamps16_31.green19 := #boGreenLampTemp;
	                #internal.lamps16_31.blue19 := #boBlueLampTemp;
	            20:
	                #internal.lamps16_31.red20 := #boRedLampTemp;
	                #internal.lamps16_31.green20 := #boGreenLampTemp;
	                #internal.lamps16_31.blue20 := #boBlueLampTemp;
	            21:
	                #internal.lamps16_31.red21 := #boRedLampTemp;
	                #internal.lamps16_31.green21 := #boGreenLampTemp;
	                #internal.lamps16_31.blue21 := #boBlueLampTemp;
	            22:
	                #internal.lamps16_31.red22 := #boRedLampTemp;
	                #internal.lamps16_31.green22 := #boGreenLampTemp;
	                #internal.lamps16_31.blue22 := #boBlueLampTemp;
	            23:
	                #internal.lamps16_31.red23 := #boRedLampTemp;
	                #internal.lamps16_31.green23 := #boGreenLampTemp;
	                #internal.lamps16_31.blue23 := #boBlueLampTemp;
	            24:
	                #internal.lamps16_31.red24 := #boRedLampTemp;
	                #internal.lamps16_31.green24 := #boGreenLampTemp;
	                #internal.lamps16_31.blue24 := #boBlueLampTemp;
	            25:
	                #internal.lamps16_31.red25 := #boRedLampTemp;
	                #internal.lamps16_31.green25 := #boGreenLampTemp;
	                #internal.lamps16_31.blue25 := #boBlueLampTemp;
	            26:
	                #internal.lamps16_31.red26 := #boRedLampTemp;
	                #internal.lamps16_31.green26 := #boGreenLampTemp;
	                #internal.lamps16_31.blue26 := #boBlueLampTemp;
	            27:
	                #internal.lamps16_31.red27 := #boRedLampTemp;
	                #internal.lamps16_31.green27 := #boGreenLampTemp;
	                #internal.lamps16_31.blue27 := #boBlueLampTemp;
	            28:
	                #internal.lamps16_31.red28 := #boRedLampTemp;
	                #internal.lamps16_31.green28 := #boGreenLampTemp;
	                #internal.lamps16_31.blue28 := #boBlueLampTemp;
	            29:
	                #internal.lamps16_31.red29 := #boRedLampTemp;
	                #internal.lamps16_31.green29 := #boGreenLampTemp;
	                #internal.lamps16_31.blue29 := #boBlueLampTemp;
	            30:
	                #internal.lamps16_31.red30 := #boRedLampTemp;
	                #internal.lamps16_31.green30 := #boGreenLampTemp;
	                #internal.lamps16_31.blue30 := #boBlueLampTemp;
	            31:
	                #internal.lamps16_31.red31 := #boRedLampTemp;
	                #internal.lamps16_31.green31 := #boGreenLampTemp;
	                #internal.lamps16_31.blue31 := #boBlueLampTemp;
	        END_CASE;
	    END_FOR;

	    IF NOT "SYS_SimulationActive" THEN
	        // Write push buttons lamps from 0 to 15
	        #readWriteData(itDeviceNumber := #itKP32DeviceNumber,
	                       uiPNIO_SysID := #uiPNIOSysID,
	                       uiSlotNumber := 1,
	                       uiSubSlotNumber := 0,
	                       bo0read_1write := TRUE,
	                       vaModuleSlotData := #internal.lamps0_15);

	        // Write push buttons lamps from 16 to 31
	        #readWriteData(itDeviceNumber := #itKP32DeviceNumber,
	                       uiPNIO_SysID := #uiPNIOSysID,
	                       uiSlotNumber := 2,
	                       uiSubSlotNumber := 0,
	                       bo0read_1write := TRUE,
	                       vaModuleSlotData := #internal.lamps16_31);
	    END_IF;

	    // Selector status to unit
	    //#unitL.from.boLeftSideSelected := #internal.panel[#PB_Configuration.itLeftSelPbID].boSelect;
	    //#unitL.from.boRightSideSelected := #internal.panel[#PB_Configuration.itRightSelPbID].boSelect;

	    //#unitR.from.boLeftSideSelected := #internal.panel[#PB_Configuration.itLeftSelPbID].boSelect;
	    //#unitR.from.boRightSideSelected := #internal.panel[#PB_Configuration.itRightSelPbID].boSelect;

	    // Equipment selection
	    #PB_Selected.itEQSelected := #NO_SELECTION;
	    IF #internal.panel[#PB_Configuration.itLoaderPbID].boSelect THEN
	        #PB_Selected.itEQSelected := #PB_Configuration.itLoaderPbID;
	    END_IF;
	    IF #internal.panel[#PB_Configuration.itGTSPbID].boSelect THEN
	        #PB_Selected.itEQSelected := #PB_Configuration.itGTSPbID;
	    END_IF;
	    IF #internal.panel[#PB_Configuration.itPressPbID].boSelect THEN
	        #PB_Selected.itEQSelected := #PB_Configuration.itPressPbID;
	    END_IF;
	    IF #internal.panel[#PB_Configuration.itSegmentsPbID].boSelect THEN
	        #PB_Selected.itEQSelected := #PB_Configuration.itSegmentsPbID;
	    END_IF;
	    IF #internal.panel[#PB_Configuration.itSqueezePbID].boSelect THEN
	        #PB_Selected.itEQSelected := #PB_Configuration.itSqueezePbID;
	    END_IF;
	    IF #internal.panel[#PB_Configuration.itExtHeatingPbID].boSelect THEN
	        #PB_Selected.itEQSelected := #PB_Configuration.itExtHeatingPbID;
	    END_IF;
	    IF #internal.panel[#PB_Configuration.itTopRingPbID].boSelect THEN
	        #PB_Selected.itEQSelected := #PB_Configuration.itTopRingPbID;
	    END_IF;
	    IF #internal.panel[#PB_Configuration.itBotRingPbID].boSelect THEN
	        #PB_Selected.itEQSelected := #PB_Configuration.itBotRingPbID;
	    END_IF;
	    IF #internal.panel[#PB_Configuration.itBeadRingPbID].boSelect THEN
	        #PB_Selected.itEQSelected := #PB_Configuration.itBeadRingPbID;
	    END_IF;
	    IF #internal.panel[#PB_Configuration.itShapingPbID].boSelect THEN
	        #PB_Selected.itEQSelected := #PB_Configuration.itShapingPbID;
	    END_IF;
	    IF #internal.panel[#PB_Configuration.itDrainPbID].boSelect THEN
	        #PB_Selected.itEQSelected := #PB_Configuration.itDrainPbID;
	    END_IF;
	    IF #internal.panel[#PB_Configuration.itVacuumPbID].boSelect THEN
	        #PB_Selected.itEQSelected := #PB_Configuration.itVacuumPbID;
	    END_IF;
	    IF #internal.panel[#PB_Configuration.itUnloaderPbID].boSelect THEN
	        #PB_Selected.itEQSelected := #PB_Configuration.itUnloaderPbID;
	    END_IF;
	    IF #internal.panel[#PB_Configuration.itUnloaderPCIPbID].boSelect THEN
	        #PB_Selected.itEQSelected := #PB_Configuration.itUnloaderPCIPbID;
	    END_IF;
	    IF #internal.panel[#PB_Configuration.itExitConvPbId].boSelect THEN
	        #PB_Selected.itEQSelected := #PB_Configuration.itExitConvPbId;
	    END_IF;
	    IF #internal.panel[#PB_Configuration.itHPUPbID].boSelect THEN
	        #PB_Selected.itEQSelected := #PB_Configuration.itHPUPbID;
	    END_IF;
	    IF #internal.panel[#PB_Configuration.itUnitPbID].boSelect THEN
	        #PB_Selected.itEQSelected := #PB_Configuration.itUnitPbID;
	    END_IF;
	    IF #internal.panel[#PB_Configuration.itPickupPbID].boSelect THEN
	        #PB_Selected.itEQSelected := #PB_Configuration.itPickupPbID;
	    END_IF;
	    IF #internal.panel[#PB_Configuration.itGymPbID].boSelect THEN
	        #PB_Selected.itEQSelected := #PB_Configuration.itGymPbID;
	    END_IF;
	    IF #internal.panel[#PB_Configuration.itLampTestPbID].boSelect THEN
	        #PB_Selected.itEQSelected := #PB_Configuration.itLampTestPbID;
	    END_IF;
	END_REGION

	REGION Side selection
	    #PB_Selected.itSideSelected := #NO_SELECTION;
	    IF #internal.panel[#PB_Configuration.itLeftSelPbID].boSelect AND #internal.panel[#PB_Configuration.itRightSelPbID].boSelect THEN
	        #PB_Selected.itSideSelected := 3;
	    ELSIF NOT #internal.panel[#PB_Configuration.itLeftSelPbID].boSelect AND #internal.panel[#PB_Configuration.itRightSelPbID].boSelect THEN
	        #PB_Selected.itSideSelected := #PB_Configuration.itRightSelPbID;
	    ELSIF #internal.panel[#PB_Configuration.itLeftSelPbID].boSelect AND NOT #internal.panel[#PB_Configuration.itRightSelPbID].boSelect THEN
	        #PB_Selected.itSideSelected := #PB_Configuration.itLeftSelPbID;
	    END_IF;
	END_REGION

